    PASSTHROUGH_SERVO_STATES.Ready :                    // Keep track    
                                                        IF jogInPB THEN
															passthroughSetpoint := 2.0 + HMIData.passthroughOffset;
															capturePassthroughPos := passthroughPosition;
															state := PASSTHROUGH_SERVO_STATES.MovePassthroughIn;
														ELSIF jogOutPB THEN
															passthroughSetpoint := 8.0 + HMIData.passthroughOffset;
															capturePassthroughPos := passthroughPosition;
															state := PASSTHROUGH_SERVO_STATES.MovePassthroughOut;
														ELSIF jogInONS.OSF OR jogOutONS.OSF THEN
															Globals.passthroughChangedFromJog := TRUE;
															pressureBarEndStopMotor.Stop();
														END_IF
														
                                                        IF _movePassthrough THEN
															passthroughTravel := ABS(passthroughPosition - (passthroughSetpoint + HMIData.passthroughOffset));
                                                            IF mustMovePassthroughOut THEN
                                                                state := PASSTHROUGH_SERVO_STATES.MovePassthroughOut;
                                                                ELSE state := PASSTHROUGH_SERVO_STATES.MovePassthroughIn;
                                                            END_IF
                                                        END_IF
                                                        IF _homeEndStop THEN
                                                            state := PASSTHROUGH_SERVO_STATES.StartHoming;
                                                        END_IF
    
    PASSTHROUGH_SERVO_STATES.Fault :   					pressureBarEndStopMotor.Stop();        
END_CASE

METHOD MovePassthrough
VAR_INPUT
    PassthroughSetting : REAL;
END_VAR
passthroughSetpoint := PassthroughSetting;
mustMovePassthroughOut := (passthroughSetpoint > passthroughPosition);
_movePassthrough := TRUE;
END_METHOD

PROPERTY Ready : BOOL
GET
Ready := _ready;
END_GET
SET
_ready := Ready;
END_SET
END_PROPERTY

PROPERTY Mode : DEVICE_MODES
GET
Mode := _mode;
END_GET
SET
_mode := Mode;
END_SET
END_PROPERTY

METHOD AckRequest
VAR_INPUT
END_VAR
_ackRequest := TRUE;
END_METHOD

METHOD HomeEndStop
VAR_INPUT
END_VAR
_homeEndStop := TRUE;
END_METHOD

END_FUNCTION_BLOCK

// FBs/Cylinders/FB_CylinderFaults
FUNCTION_BLOCK FB_CylinderFaults
VAR_INPUT
	enable : BOOL;
	extendCommand : BOOL;
	extendedInput : BOOL;
	retractCommand : BOOL;
	retractedInput : BOOL;
	faultTime : TIME := T#2500ms;
END_VAR
VAR_OUTPUT
	failToExtend : BOOL;
	failToRetract : BOOL;
END_VAR
VAR
	extendFaultTimer : Standard.TON;
	retractFaultTimer : Standard.TON;
END_VAR
VAR_IN_OUT
END_VAR

extendFaultTimer(PT := faultTime, Q => failToExtend);
retractFaultTimer(PT := faultTime, Q => failToRetract);
IF enable THEN
	IF extendCommand THEN
		retractFaultTimer.IN := FALSE;
		extendFaultTimer.IN := NOT extendedInput;
	ELSIF retractCommand THEN
		extendFaultTimer.IN := FALSE;
		retractFaultTimer.IN := NOT retractedInput;
	ELSE
		retractFaultTimer.IN := FALSE;
		extendFaultTimer.IN := FALSE;
	END_IF
ELSE
	retractFaultTimer.IN := FALSE;
	extendFaultTimer.IN := FALSE;
END_IF

END_FUNCTION_BLOCK

// FBs/FB_HMILight
FUNCTION_BLOCK FB_HMILight
VAR_INPUT
END_VAR
VAR_OUTPUT
	lightOutput : BOOL;
END_VAR
VAR
	_turnOn : BOOL;
	_blinkFast : BOOL;
	_blinkSlow : BOOL;
	blinker : OSCAT_BASIC.PWM_DC := (F := 1, DC := 0.5);
	slowBlinkSec : REAL := 1;
	fastBlinkSec : REAL := 0.5;
END_VAR

IF _blinkFast THEN
	blinker.F := fastBlinkSec;
ELSIF _blinkSlow THEN 
	blinker.F := slowBlinkSec;
END_IF
	
blinker(F:= , DC:= , Q=> );

lightOutput := _turnOn OR (blinker.Q AND (_blinkFast OR _blinkSlow));

METHOD BlinkSlow
VAR_INPUT
END_VAR
_blinkFast := FALSE;
_blinkSlow := TRUE;
_turnOn := FALSE;
END_METHOD

METHOD BlinkFast
VAR_INPUT
END_VAR
_blinkFast := TRUE;
_blinkSlow := FALSE;
_turnOn := FALSE;
END_METHOD

METHOD TurnOff
VAR_INPUT
END_VAR
_blinkFast := FALSE;
_blinkSlow := FALSE;
_turnOn := FALSE;
END_METHOD

METHOD TurnOn
VAR_INPUT
END_VAR
_blinkFast := FALSE;
_blinkSlow := FALSE;
_turnOn := TRUE;
END_METHOD

END_FUNCTION_BLOCK

// FBs/Components/FillerFB
FUNCTION_BLOCK FillerFB EXTENDS BaseComponentFB IMPLEMENTS IComponentStatus
VAR_INPUT
	fillerTrigger : BOOL;
	activateFiller : BOOL;
	fillerOK : BOOL;
	dropTime : REAL;
END_VAR
VAR_OUTPUT
	state : FILLER_STATES;
	fillerModeActive : BOOL;
	waitingForFiller : BOOL;
	cycleBagRequest : BOOL;
	cycleBaggerToActivateFiller : Warning;
	notReady : FB_Fault(name := 'Not Ready');
END_VAR
VAR
	_baggerCycleInitiated : BOOL;
    _baggerCycledAndReady : BOOL;
	fillerRequestedCycle : BOOL;
	fillerTrigONS : FB_ONS;
	dropTimer : Standard.TON;
END_VAR
	
VAR_IN_OUT
END_VAR

//    Function Block: FillerFB
//    Description: Filler state machine
//    Created by: Ben Hess
//    Created Date: October 16th, 2019
SUPER^();
dropTimer(PT := TO_TIME(dropTime * 1000));
IF resetONS.Q OR HMIData.faultActive OR NOT enable OR NOT activateFiller THEN
	state := FILLER_STATES.Idle;
	fillerRequestedCycle := FALSE;
	cycleBaggerToActivateFiller.active := FALSE;
	waitingForFiller := FALSE;
	cycleBagRequest := FALSE;
	_baggerCycledAndReady := FALSE;
	_baggerCycleInitiated := FALSE;
	dropTimer.IN := FALSE;
END_IF

IF NOT fillerOK AND enable AND activateFiller THEN
	notReady.Trigger();
END_IF

fillerTrigONS(CLK := fillerTrigger);
IF fillerTrigONS.OSR THEN
	fillerRequestedCycle := TRUE;
END_IF

CASE state OF
	FILLER_STATES.Idle :							IF (activateFiller AND enable) AND NOT HMIData.faultActive THEN
														state := FILLER_STATES.CycleBaggerToActiveFiller;
													END_IF
	
	FILLER_STATES.CycleBaggerToActiveFiller :		// Operator must cycle a bag out first to guarentee bag open and ready for filler
													cycleBaggerToActivateFiller.active := TRUE;
													
													IF _baggerCycledAndReady THEN
														cycleBaggerToActivateFiller.active := FALSE;
														_baggerCycledAndReady := FALSE;
														fillerRequestedCycle := FALSE;
														state := FILLER_STATES.WaitingForFiller;
													END_IF
	
	FILLER_STATES.WaitingForFiller :				// Waiting for filler trigger to initiate cycle
													waitingForFiller := TRUE;
													IF fillerRequestedCycle THEN
														waitingForFiller := FALSE;	
														//IF NOT HMIData.baggerInhibited.active THEN
															fillerRequestedCycle := FALSE;
															state := FILLER_STATES.Dropping;	
														//END_IF
													END_IF
													
	FILLER_STATES.Dropping :						// Filler is dropping product
													dropTimer.IN := TRUE;
													IF dropTimer.Q THEN
														IF NOT HMIData.baggerInhibited.active THEN
															dropTimer.IN := FALSE;
															cycleBagRequest := TRUE;
															state := FILLER_STATES.BaggerCycling;	
														END_IF
													END_IF
	
	FILLER_STATES.BaggerCycling :					// Wait for bag to open 
													IF _baggerCycleInitiated THEN
														_baggerCycleInitiated := FALSE;
														cycleBagRequest := FALSE;
													END_IF
													
													IF _baggerCycledAndReady THEN
														_baggerCycledAndReady := FALSE;
														state := FILLER_STATES.WaitingForFiller;
													END_IF
	
	FILLER_STATES.Fault :
	
END_CASE

METHOD BaggerCycledAndReady : BOOL
VAR_INPUT
END_VAR
_baggerCycledAndReady := TRUE;
END_METHOD

PROPERTY Ready : BOOL
SET
_ready := Ready;
END_SET
GET
Ready := _ready;
END_GET
END_PROPERTY

METHOD BaggerCycleInitiated : BOOL
VAR_INPUT
END_VAR
_baggerCycleInitiated := TRUE;
END_METHOD

PROPERTY Mode : DEVICE_MODES
SET
_mode := Mode;
END_SET
GET
Mode := _mode;
END_GET
END_PROPERTY

METHOD Reset : BOOL
VAR_INPUT
END_VAR
SUPER^.Reset();
END_METHOD

END_FUNCTION_BLOCK

// FBs/Components/MurrIOFB
FUNCTION_BLOCK MurrIOFB EXTENDS BaseComponentFB IMPLEMENTS IComponentStatus
VAR_INPUT
	headNodeEnabled : BOOL;
	guardNodeEnabled : BOOL;
	printerNodeEnabled : BOOL;
	dischargeNodeEnabled : BOOL;
	auxIONodeEnabled : BOOL;
	configVersion : CONFIG_VERSIONS;
	ptrMachineOptionsManagementOutputs : POINTER TO BYTE;
	ptrSystemStatusInputs : POINTER TO BYTE;
END_VAR
VAR_OUTPUT
	commFailController : FB_Fault(name := 'Communication Fail - Bus Master to Controller');
	commFailNode : FB_Fault(name := 'Communication Fail - Bus Master to I/O Node');
	configActive : Warning;	// I/O Configuration Active, please wait
	ok : BOOL; 		// I/O Configuration and Communication good
END_VAR
VAR
	systemStatusINT : INT;
	systemStatusState : MURR_SYSTEM_STATES;
	MOMConfigLast : BYTE;
	restartBusnodePulse : MonostableMultivibratorFB;
END_VAR
	
VAR_IN_OUT

END_VAR

//    Function Block: MurrIOFB
//    Description: Alarms, faults, configuration of the Murr Cube67+ Bus Node
//    Created by: Ben Hess
//    Created Date: October 16th, 2019
SUPER^();

// Set bit 33 to true for 1 second to reset nodes
restartBusnodePulse.DwellSetting := 1000;
restartBusnodePulse(Q => ptrMachineOptionsManagementOutputs[4].1);

// Exit this FB if invaild pointers set
IF ptrMachineOptionsManagementOutputs = 0 OR ptrSystemStatusInputs = 0 THEN
	RETURN;
END_IF

// MOM config - MOM bits are counted from Slot 001 to 4xx and are counted based on the "Maximium" configuration hard coded in the bus master
// Here we can select which verison of code we have in order to utilize MOM correctly if we add additional modules in the future.
CASE configVersion OF
	CONFIG_VERSIONS.V_1_1 :		//
									ptrMachineOptionsManagementOutputs[0].0 := NOT headNodeEnabled;
									ptrMachineOptionsManagementOutputs[0].1 := NOT guardNodeEnabled;
									ptrMachineOptionsManagementOutputs[0].2 := NOT dischargeNodeEnabled;
									ptrMachineOptionsManagementOutputs[0].3 := NOT printerNodeEnabled;
									ptrMachineOptionsManagementOutputs[0].4 := FALSE;
									
								

	CONFIG_VERSIONS.V_1_2, CONFIG_VERSIONS.V_1_3,CONFIG_VERSIONS.V_1_4 : 		// Added aux IO to 1.2 and BCV trigger to 1.3
									ptrMachineOptionsManagementOutputs[0].0 := NOT headNodeEnabled;
									ptrMachineOptionsManagementOutputs[0].1 := NOT guardNodeEnabled;
									ptrMachineOptionsManagementOutputs[0].2 := NOT auxIONodeEnabled;
									ptrMachineOptionsManagementOutputs[0].3 := NOT dischargeNodeEnabled;
									ptrMachineOptionsManagementOutputs[0].4 := NOT printerNodeEnabled;
END_CASE


// Run config if IO bus node is waiting on config
systemStatusINT := ptrSystemStatusInputs^;
systemStatusState := systemStatusINT;

// Prevent a IO node reset on boot for no reason
IF Globals.firstScan THEN
	MOMConfigLast := ptrMachineOptionsManagementOutputs[0];
END_IF

// Trigger fault for node not present, or node seen where one shouldn't be 
IF systemStatusState = MURR_SYSTEM_STATES.No_Comm_To_Configured_Node THEN
	commFailNode.Trigger();
END_IF

// A 0 at system state indicates comm fail to controller
IF systemStatusState = 0 THEN
	commFailController.Trigger();
END_IF

// Alert user to MOM config active
IF systemStatusState = MURR_SYSTEM_STATES.Waiting_For_MOM OR
	systemStatusState = MURR_SYSTEM_STATES.Configuring_MOM OR
	systemStatusState = MURR_SYSTEM_STATES.Internal_Comm_Disabled
THEN
	configActive.active := TRUE;
ELSE
	configActive.active := FALSE;
END_IF

// I/O Block is OK only in this state, otherwise we can't trust any I/O coming back
ok := (systemStatusState = MURR_SYSTEM_STATES.Internal_Comm_OK);

CASE systemStatusState OF

	
	MURR_SYSTEM_STATES.Waiting_For_MOM: 			// Bit 32 is Configure MOM bit
													ptrMachineOptionsManagementOutputs[4].0 := TRUE;
													ptrMachineOptionsManagementOutputs[4].1 := FALSE;
													
	
	MURR_SYSTEM_STATES.Configuring_MOM : 			//
													ptrMachineOptionsManagementOutputs[4].0 := FALSE;
													
											

														
											
ELSE
													ptrMachineOptionsManagementOutputs[4].0 := FALSE;
													//IF config changes here, send it down after restarting
													IF ptrMachineOptionsManagementOutputs[0] <> MOMConfigLast THEN
														restartBusnodePulse.Trigger();
														MOMConfigLast := ptrMachineOptionsManagementOutputs[0];
													END_IF
END_CASE

PROPERTY Mode : DEVICE_MODES
GET
Mode := _mode;
END_GET
SET
_mode := Mode;
END_SET
END_PROPERTY

PROPERTY Ready : BOOL
GET
Ready := _ready;
END_GET
SET
_ready := Ready;
END_SET
END_PROPERTY

END_FUNCTION_BLOCK

// FBs/Components/FunnelFB
FUNCTION_BLOCK FunnelFB EXTENDS BaseComponentFB
VAR_INPUT
	sensorsInstalled : BOOL;							// Are open/closed sensors installed?
	openSensor : BOOL;									// Open sensor input
	closedSensor : BOOL;								// Closed sensor input
END_VAR	
VAR_OUTPUT
	opened : BOOL;										// Funnel Opened status
	closed : BOOL;										// Funnel Closed status
	closeOutput : BOOL;									// Map to physical close output
	openOutput : BOOL;									// Map to physical open output
	failToOpen : FB_Fault(name := 'Failed to Open');	// Failed to Open fault
	failToClose : FB_Fault(name := 'Failed to Close');	// Failed to Close fault
END_VAR
VAR
	_delayTimeInMS : UINT; 								// Delay before open in mS
	_closeReq : BOOL;									// Close reqested from CloseNow()
	_openReq : BOOL;									// Open requested from OpenNow()
	openDelayTimer : Standard.TON;						// Open delay timer
	openingTimer : Standard.TON;						// Opening timer
	closingTimer : Standard.TON;						// Closing timer
	faultTimer : FB_CylinderFaults;						// Fault timer for open/close faults
END_VAR

//    Function Block: FunnelFB
//    Description: Funnel
//    Created by: Ben Hess
//    Created Date: November 18th, 2019

IF _reset THEN
	_openReq := FALSE;
	_closeReq := FALSE;
	openingTimer.IN := FALSE;
	closingTimer.IN := FALSE;
	openDelayTimer.IN := FALSE;
END_IF

// Setup timers
openDelayTimer();
openingTimer();
closingTimer();

// Use opening/closing timers for debounce if sensors enabled
// or for actual opening/closing time after command to move if disabled
IF sensorsInstalled THEN
	openingTimer.IN := openSensor;
	closingTimer.IN := closedSensor;
ELSE
	openingTimer.IN := openOutput;
	closingTimer.IN := closeOutput;
END_IF

// Set open/closed status of funnel
opened := openingTimer.Q;
closed := closingTimer.Q;


// Set physical outputs depending on command
IF enable THEN
	IF _closeReq THEN
		closeOutput := TRUE;
		openOutput := FALSE;
		_closeReq := FALSE;
	ELSIF _openReq THEN
		openDelayTimer.IN := TRUE;
		closeOutput := FALSE;
		openOutput := openDelayTimer.Q;
		_openReq := FALSE;
	END_IF
ELSE
	// Turn everything off if disabled
	closeOutput := FALSE;
	openOutput := FALSE;
	_openReq := FALSE;
	_closeReq := FALSE;
	openingTimer.IN := FALSE;
	closingTimer.IN := FALSE;
	openDelayTimer.IN := FALSE;
END_IF

// Fault timer for failed to reach open/closed sensors
faultTimer(
	enable:= THIS^.enable AND sensorsInstalled, 
	extendCommand:= closeOutput, 
	extendedInput:= closedSensor, 
	retractCommand:= openOutput, 
	retractedInput:= openSensor, 
	faultTime:= T#1S, 
	failToExtend=> failToClose.faultTrigger, 
	failToRetract=> failToOpen.faultTrigger);
	
SUPER^();

PROPERTY DelaySetting : REAL
GET
DelaySetting := TO_REAL(openDelayTimer.PT ) / 1000;
END_GET
SET
openDelayTimer.PT := TO_TIME(DelaySetting * 1000);
END_SET
END_PROPERTY

METHOD CloseNow : BOOL
VAR_INPUT
END_VAR
_closeReq := TRUE;
END_METHOD

PROPERTY OpeningTime : REAL
SET
openingTimer.PT := TO_TIME(OpeningTime * 1000);
END_SET
GET
OpeningTime := TO_REAL(openingTimer.PT) / 1000;
END_GET
END_PROPERTY

METHOD OpenNow : BOOL
VAR_INPUT
END_VAR
_openReq := TRUE;
END_METHOD

PROPERTY ClosingTime : REAL
GET
ClosingTime := TO_REAL(closingTimer.PT) / 1000;
END_GET
SET
closingTimer.PT := TO_TIME(ClosingTime * 1000);
END_SET
END_PROPERTY

END_FUNCTION_BLOCK

// FBs/Components/BarcodeReaderFB
FUNCTION_BLOCK BarcodeReaderFB EXTENDS BaseComponentFB
VAR_INPUT
	feedSpeed : REAL;
	positionOffset : REAL;
	distanceToScan : REAL;
	readGoodInput : BOOL;
	badReadFaultCountSetting : UDINT;
END_VAR	
VAR_OUTPUT
	triggerScannerOutput : BOOL;
	xBusy : BOOL;
	xDone : BOOL;
	currentGoodReadCount : UDINT;
	currentBadReadCount : UDINT;
	barcodeFault : BOOL;
END_VAR
VAR
	_goodRead : BOOL;
	_badread : BOOL;
	_trigger : BOOL;
	state : BCR_STATES;
	waitForReadTimer : Standard.TON;
	positionOffsetDelay : Standard.TON;
END_VAR
VAR CONSTANT
	MILLISECONDS_IN_SECOND : INT := 1000;
END_VAR

//    Function Block: BarcodeReaderFB
//    Description: Trigger the barcode verifier and receive a "Barcode OK" signal, or nothing which indicates no read.
//    Created by: Ben Hess
//    Created Date: January 29th, 2020

// Setup timers for reading offset and scanning distance
IF positionOffset > 0 THEN
	positionOffsetDelay(PT := TO_TIME(MILLISECONDS_IN_SECOND / (feedSpeed / positionOffset)) + T#120ms);
ELSE
	positionOffsetDelay(PT := T#0S);
END_IF

IF distanceToScan > 0 THEN
	waitForReadTimer(PT := TO_TIME(MILLISECONDS_IN_SECOND / (feedSpeed / distanceToScan)));
ELSE
	waitForReadTimer(PT := T#0S);
END_IF

IF _reset OR NOT enable THEN
	//
	state := BCR_STATES.Idle;
	barcodeFault := FALSE;
END_IF

CASE state OF
	
	BCR_STATES.Idle:				// Wait for trigger
									triggerScannerOutput := FALSE;
									waitForReadTimer.IN := FALSE;
									positionOffsetDelay.IN := FALSE;
									
									xBusy := FALSE;
									IF _trigger THEN
										state := BCR_STATES.WaitForOffset;
										positionOffsetDelay.IN := TRUE;
										xBusy := TRUE;
										xDone := FALSE;
									END_IF
									
									_trigger := FALSE;
									
	BCR_STATES.WaitForOffset: 		// Wait for offset to trigger read
									IF positionOffsetDelay.Q THEN
										state := BCR_STATES.TriggerReader;
										positionOffsetDelay.IN := FALSE;
									END_IF
									
	BCR_STATES.TriggerReader:		// Trigger the reader and then move to waiting state for result
									triggerScannerOutput := TRUE;
									waitForReadTimer.IN := TRUE;
									state := BCR_STATES.WaitingForResult;
									
	
	BCR_STATES.WaitingForResult:	// Wait for delayToCheckReadStatus timer.  If it times out we did not get a good read
									IF readGoodInput THEN
										_goodRead := TRUE;
										_badread := FALSE;
										currentGoodReadCount := currentGoodReadCount + 1;
										currentBadReadCount := 0;
										xDone := TRUE;
										state := BCR_STATES.Idle;
									ELSIF waitForReadTimer.Q THEN
										_goodRead := FALSE;
										_badread := TRUE;
										currentGoodReadCount := 0;
										currentBadReadCount := currentBadReadCount + 1;
										IF badReadFaultCountSetting > 0 THEN
											IF currentBadReadCount >= badReadFaultCountSetting THEN
												barcodeFault := TRUE;
											END_IF
										END_IF
										xDone := TRUE;
										state := BCR_STATES.Idle;
									END_IF
	
	BCR_STATES.Resetting:
	
END_CASE

SUPER^();

METHOD Trigger : BOOL
VAR_INPUT
END_VAR
_trigger := TRUE;
END_METHOD

PROPERTY BadRead : BOOL
SET
END_SET
GET
END_GET
END_PROPERTY

PROPERTY GoodRead : BOOL
GET
END_GET
SET
END_SET
END_PROPERTY

END_FUNCTION_BLOCK

// FBs/Components/KeyenceL20FB/KeyenceNL20FB
FUNCTION_BLOCK KeyenceNL20FB EXTENDS BaseComponentFB IMPLEMENTS IComponentStatus
VAR_INPUT
	ptrEIPInputs : POINTER TO WORD;
	ptrEIPOutputs : POINTER TO WORD;
	triggerInput : BOOL;
END_VAR
VAR_OUTPUT
	lastReadData : STRING[100];
	xBusy : BOOL;
	xDone : BOOL;
	goodRead : BOOL;
	badRead : BOOL;
END_VAR
VAR
	error : BOOL;
	readDataUpdateAvailable : BOOL;
	readDataUpdateComplete : BOOL;
	bufferOverflowError : BOOL;
	generalError : BOOL;
	bcvBusy : BOOL;
	readingComplete : BOOL;
	in1Status : BOOL;
	in2Status : BOOL;
	out1Status : BOOL;
	out2Status : BOOL;
	out3Status : BOOL;
	out4Status : BOOL;
	errorCode : UINT;
	readDataReadyCount : UINT;
	readDataUpdateCount : UINT;
	readDataLength : UINT;
	readData : POINTER TO STRING[100];
	
	readDataUpdatePermitted : BOOL;
	errorAndBufferClear : BOOL;
	readingStartRequest : BOOL;
	readingCompleteAck : BOOL;
	bankNumber : UINT;
	
	state : eKeyenceLN20FB_States;
	triggerONS : FB_ONS;
	readingCompleteTrigger : MonostableMultivibratorFB();
END_VAR
	
VAR_IN_OUT

END_VAR

//    Function Block: KeyenceL20FB
//    Description: Alarms, faults, configuration of the Keyence L-N20 barcode scanner base
//    Created by: Ben Hess
//    Created Date: Feb 28th, 2020


// Exit FB if pointers are invalid
IF ptrEIPInputs = 0 OR ptrEIPOutputs = 0 THEN
	RETURN;
END_IF
triggerONS(CLK := triggerInput);

readingCompleteTrigger.DwellSetting := 500;
readingCompleteTrigger(Q => readingCompleteAck);
// Map statuses to friendly variables
error := ptrEIPInputs[0].0;
readDataUpdateAvailable := ptrEIPInputs[0].1;
readDataUpdateComplete := ptrEIPInputs[0].2;
bufferOverflowError := ptrEIPInputs[0].6;
generalError := ptrEIPInputs[0].7;
bcvBusy := ptrEIPInputs[0].8;

readingComplete := ptrEIPInputs[1].0;

in1Status := ptrEIPInputs[2].0;
in2Status := ptrEIPInputs[2].1;
out1Status := ptrEIPInputs[2].4;
out2Status := ptrEIPInputs[2].5;
out3Status := ptrEIPInputs[2].6;
out4Status := ptrEIPInputs[2].7;

errorCode := ptrEIPInputs[16];

readDataReadyCount := ptrEIPInputs[18];
readDataUpdateCount := ptrEIPInputs[19];

readDataLength := ptrEIPInputs[21];
readData := ADR(ptrEIPInputs[22]);


IF resetONS.Q THEN
	state := eKeyenceLN20FB_States.Reset;
END_IF



CASE state OF
	eKeyenceLN20FB_States.Idle: 			//
											IF readingComplete THEN
													readingCompleteTrigger.Trigger();
												END_IF
											IF triggerONS.OSR THEN
												readingStartRequest := TRUE;
												xBusy := TRUE;
												xDone := FALSE;
												badRead := FALSE;
												goodRead := FALSE;
												lastReadData := '---Read in Progress---';
												state := eKeyenceLN20FB_States.WaitForStatus;
											END_IF

	eKeyenceLN20FB_States.WaitForStatus:	//
											IF readingComplete OR NOT triggerInput THEN
												state := eKeyenceLN20FB_States.SetStatus;
												readingStartRequest := FALSE;
												IF readingComplete THEN
													readingCompleteTrigger.Trigger();
												END_IF
												
											END_IF
	
	eKeyenceLN20FB_States.SetStatus:		// Set the current read status and string
											// If trigger input goes away or barcode error seen set bad read
											IF NOT triggerInput OR out2Status THEN
												badRead := TRUE;
												goodRead := FALSE;
												state := eKeyenceLN20FB_States.WaitForReadClear;
												IF out2Status THEN
													lastReadData := '---BAD READ---';
												ELSE
													lastReadData := '---NO READ---';
												END_IF
											ELSIF out1Status THEN
												goodRead := TRUE;
												badRead := FALSE;
												// Strip terminating char (0x0D) from string to get clean read barcode
												lastReadData := LEFT(readData^, readDataLength - 1);
												state := eKeyenceLN20FB_States.WaitForReadClear;
											END_IF
											
	eKeyenceLN20FB_States.WaitForReadClear:	//
											IF readingComplete THEN
												readingCompleteTrigger.Trigger();
											END_IF
											IF NOT readingComplete THEN
												xBusy := FALSE;
												xDone := TRUE;
												state := eKeyenceLN20FB_States.Idle;
											END_IF 									

	eKeyenceLN20FB_States.Reset: 			//
											IF readingComplete THEN
												readingCompleteTrigger.Trigger();
											END_IF
											
												readingStartRequest := FALSE;
												xBusy := FALSE;
												xDone := FALSE;
												badRead := FALSE;
												goodRead := FALSE;
												state := eKeyenceLN20FB_States.Idle;
											
END_CASE	

// Outputs to barcode verifier
ptrEIPOutputs[0].1 :=  readDataUpdatePermitted;
ptrEIPOutputs[0].7 :=  errorAndBufferClear;
ptrEIPOutputs[0].8 := readingStartRequest;
ptrEIPOutputs[1].0 := readingCompleteAck;
ptrEIPOutputs[2] := bankNumber;

// Call to super FB.
SUPER^();

PROPERTY Ready : BOOL
SET
_ready := Ready;
END_SET
GET
Ready := _ready;
END_GET
END_PROPERTY

PROPERTY Mode : DEVICE_MODES
SET
_mode := Mode;
END_SET
GET
Mode := _mode;
END_GET
END_PROPERTY

END_FUNCTION_BLOCK

// FBs/Components/EZFeedFB/EZFeedFB
FUNCTION_BLOCK EZFeedFB EXTENDS BaseComponentFB IMPLEMENTS IComponentStatus
VAR_INPUT
	baggerFaulted : BOOL;
	enableEZFeed : BOOL;					// Enable EZFeed conveyor (In Use)
	continuousModeEnable : BOOL; 			// 0 = indexing mode, 1 = continuous mode
	partsCountingModeEnable : BOOL;			// 0 = Flight counting only, 1 = Parts counting (requires sensor or light curtains)
	flightPresentSensor : BOOL;				// Flight present 
	partPresentSensor : BOOL;				// Part present/dropping (photoeye, light curtain, etc)
	waitingForFiller : BOOL;				// Waiting for Filler signal from bagger
	indexDwellSetting : REAL;				// Indexing dwell setting
	flightTarget : DINT;					// For Flight counting mode, target flights before starting cycle
	partsTarget : DINT;						// For Parts counting mode, target parts before starting cycle
	emptyPartsWarningSetting : DINT;		// For Parts counting mode, setting of empty flights counted before warning issued
	restartFromEmptyParts : BOOL;			// Restart EZFeed after starvation/empty parts. Usually cycle start button
END_VAR
VAR_OUTPUT
	state : EZFEED_STATES;					// State machine
	runVFD : BOOL;							// Run VFD output
	flightCount : DINT;						// Actual flight count
	partsCount : DINT;						// Actual parts count
	emptyPartsWarningCount : DINT;			// Actual empty flights count
	EZFeedDone : BOOL;						// EZFeed done - cycle bagger
	emptyPartsWarning : BOOL;				// Parts starved
END_VAR
VAR
	indexDwellTimer : TON;
	flightPresentONS : FB_ONS;
	partPresentONS : FB_ONS;
END_VAR
	
VAR_IN_OUT
END_VAR

//    Function Block: EZFeedFB
//    Description: EZFeed state machine
//    Created by: Ben Hess
//    Created Date: December 3rd, 2020


// Run parent FB
SUPER^();

// Resetting 
IF resetONS.Q OR baggerFaulted OR NOT enable OR NOT enableEZFeed THEN
	state := EZFEED_STATES.Idle;
	runVFD := FALSE;
	EZFeedDone := FALSE;
	flightCount := 0;
	partsCount := 0;
	emptyPartsWarningCount := 0;
END_IF

// Timer for indexing dwell
indexDwellTimer(PT := TO_TIME(indexDwellSetting * 1000), IN := state = EZFEED_STATES.IndexDwell);

flightPresentONS(CLK := flightPresentSensor);
partPresentONS(CLK := partPresentSensor);

// Parts Counting logic
IF partsCountingModeEnable AND (state = EZFEED_STATES.IndexingFlightMode OR state = EZFEED_STATES.IndexDwell) THEN
	// Count flights for empty parts watchdog timer
	IF flightPresentONS.OSR THEN
		emptyPartsWarningCount := emptyPartsWarningCount + 1;
	END_IF
	
	IF partPresentONS.OSF THEN
		emptyPartsWarningCount := 0;
		partsCount := partsCount + 1;
	END_IF
	
END_IF

CASE state OF
	
	EZFEED_STATES.Idle :						// When filler reports as waiting for filler, start indexing the EZFeed
												IF enableEZFeed AND waitingForFiller THEN
													IF partsCountingModeEnable THEN
														state := EZFEED_STATES.IndexingPartsMode;
													ELSE
														state := EZFEED_STATES.IndexingFlightMode;
													END_IF
													
												END_IF
	
	EZFEED_STATES.IndexingPartsMode :			// Check parts count and start bagger if count reached
												IF partsCount >= partsTarget THEN
													partsCount := 0;
													runVFD := FALSE;
													EZFeedDone := TRUE;
													state := EZFEED_STATES.WaitForBaggerCycleComplete;
												ELSE
													// Dwell at each flight for indexing mode
													IF NOT continuousModeEnable THEN
														runVFD := FALSE;
														state := EZFEED_STATES.IndexDwell;
													END_IF
												END_IF

												
		
	EZFEED_STATES.IndexingFlightMode :			// Run the VFD until flight seen. Keep going until target reached in Continuous mode or stop for dwell time in indexing mode
												runVFD := TRUE;
												IF flightPresentONS.OSR THEN
													flightCount := flightCount + 1;
													// Check flight count and start bagger if count reached
													IF flightCount >= flightTarget THEN
														runVFD := FALSE;
														EZFeedDone := TRUE;
														flightCount := 0;
														state := EZFEED_STATES.WaitForBaggerCycleComplete;
													ELSE
														// Dwell at each flight for indexing mode
														IF NOT continuousModeEnable THEN
															runVFD := FALSE;
															state := EZFEED_STATES.IndexDwell;
														END_IF
													END_IF
												END_IF
												
	EZFEED_STATES.IndexDwell :					// Dwell at each flight for indexing mode
												IF indexDwellTimer.Q THEN
													IF partsCountingModeEnable THEN
														IF partsCount >= partsTarget THEN
															partsCount := 0;
															EZFeedDone := TRUE;
															state := EZFEED_STATES.WaitForBaggerCycleComplete;
														ELSE
															state := EZFEED_STATES.IndexingPartsMode;
														END_IF
													ELSE
														state := EZFEED_STATES.IndexingFlightMode;
													END_IF
												END_IF
												
	EZFEED_STATES.WaitForBaggerCycleComplete :	// Once bagger cycle is complete then resume indexing
												IF waitingForFiller THEN
													IF partsCountingModeEnable THEN
														state := EZFEED_STATES.IndexingPartsMode;
													ELSE
														state := EZFEED_STATES.IndexingFlightMode;
													END_IF
												END_IF
								
	EZFEED_STATES.PartsStarved:					//
												
									
	EZFEED_STATES.Fault :						//
												

END_CASE

PROPERTY Mode : DEVICE_MODES
SET
_mode := Mode;
END_SET
GET
Mode := _mode;
END_GET
END_PROPERTY

PROPERTY Ready : BOOL
GET
Ready := _ready;
END_GET
SET
_ready := Ready;
END_SET
END_PROPERTY

METHOD Reset : BOOL
VAR_INPUT
END_VAR
SUPER^.Reset();
END_METHOD

END_FUNCTION_BLOCK

// FBs/GetTime
FUNCTION_BLOCK GetTime
VAR_INPUT
END_VAR
VAR_OUTPUT
    currentDateAndTime : DATE_AND_TIME;
    
END_VAR
VAR
    iState                    : INT;
    udiUtcTime             : UDINT;
    udiUtcTimeLocal     : UDINT;
    strTimeDate         : SYSTIMEDATE;
    strTimeDateLocal     : SYSTIMEDATE;
    dtDateTimeUTC        : DATE_AND_TIME;
    timeLeftTime        : TIME;
    timeLeftDWORD        : DWORD;
    dDateUTC            : DATE;
    todTimeOfDayUTC        : TOD;
    
    tSysStartTime        : TIME;
    systimeStartNano    : SYSTIME;
    udiStartTimeResult    : UDINT;
    
    udiResult             : UDINT;
    
    
    GetDateAndTime            : DTU.GetDateAndTime;
    SetTimeZoneInformation    : DTU.SetTimeZoneInformation;
    
    dtCurrent                : DATE_AND_TIME;
    dtConcated                : DATE_AND_TIME;
    eWeekday                 : RTCLK.WEEKDAY;
    uiYear                     : UINT;
    uiMonth                     : UINT;
    uiDay                     : UINT;
    uiHour                     : UINT;
    uiMinute                 : UINT;
    uiSecond                 : UINT;
        
    dtuError                : DTU.ERROR;
END_VAR

CASE iState OF

    0:    
        iState:= 1;
        
    1:  // retrieves the target date and time, including the timezone information which was set before
        GetDateAndTime( xExecute:= TRUE);
        IF GetDateAndTime.xDone THEN
            dtCurrent:= GetDateAndTime.dtDateAndTime;
            GetDateAndTime(xExecute:= FALSE);
			currentDateAndTime := dtCurrent;
            //timeLeft := TIME_TO_DT(DT_TO_TIME(targetDate) - DT_TO_TIME(dttarget));
            iState:= 2;
        END_IF
        IF GetDateAndTime.xError THEN
            GetDateAndTime(xExecute:= FALSE);
            iState:= 32767;
        END_IF
    
    2: (*set a spedific date and time --> returns a variable of type DATE_AND_TIME 
         DateConcat --> set only date information --> returns a variable of type DATE
         TODConcat  --> set only the time information  --> returns a variable of TOD (Time of day) *)
        IF dtuError = 0 THEN
            iState := 3;
        ELSE
            iState := 32767;
        END_IF
        
    3:  (*a DATE_AND_TIME variable is splitted in its parts, like year, month, day etc.
            DateSplit --> the same function for a DATE variable
            TODSplit  --> the same function for a TOD variable *)

            
        IF dtuError = 0 THEN
            iState:= 1;
        ELSE
            iState:= 32767;
        END_IF
        
    32767: ; //error

END_CASE

END_FUNCTION_BLOCK

// FBs/FunctionalAreas/FB_MOABHead_Electric
FUNCTION_BLOCK FB_MOABHead_Electric EXTENDS BaseComponentFB
VAR_INPUT
    motorizedSealFlattenersMode : DEVICE_MODES := DEVICE_MODES.Auto;
    electricPressureBarMode : DEVICE_MODES := DEVICE_MODES.Auto;
	vacuumPickerMode : DEVICE_MODES;
    startCycle : BOOL;
    bagDeliveryMode : DEVICE_MODES;        // Mode of bag delivery system
    printerMode : DEVICE_MODES;        // Mode of printer
	passthroughMode : DEVICE_MODES;
    batchSetting : DINT;            // Batch setpoint
    batchCount : DINT;                // Actual batch cycles
    enableBatch : BOOL;                // Enable Batch Mode
    enableBatchONS : F_TRIG;
	passthroughSetting : REAL;
    passthroughSettingLast : REAL;
	bagDropDelay : UINT := 1000;
END_VAR
VAR_OUTPUT
    readyToRun : BOOL;
    state : HEAD_STATES;
    sealAndSeparateSubState : SEAL_SEPARATE_STATES;
    releaseAndFeedSubState : RELEASE_FEED_STATES;
    openBagSubState : BAG_OPEN_ASSIST_STATES;
	finishCycleSubState : FINISH_CYCLE_STATES;
END_VAR
VAR
    motorizedSealFlatteners : MotorizedSealFlattenersFB_BagFeed();
	msfVerticalAxis : FB_ThreePositionCylinder();
    pressureBar : FB_MotorizedPressureBar();
	IBD : FB_MotorizedIBD();
	sealBarTempSensor : FB_IFMTempSensor();
	sealBarHeater : FB_TempController();
    startCycleONS : R_TRIG;
	enableBagOpen : BOOL;
	enableLoadPlate : BOOL;
	enableHeater : BOOL;
	enableIBDDeflate : BOOL;
	enableIBDEject : BOOL;
	enableLabelSideUp : BOOL := TRUE;
	factoryTestModeKeepCycling : BOOL;
	autoModeKeepCycling : BOOL;
	autoModeKeepCyclingTimer : Standard.TON;
    bagDelivery : BagDeliveryFB();
    //zebraPrinter : PrinterFB;            //Printer Test Rig
	zebraPrinter : PrinterFB_Mode2;
	sealTimer : Standard.TON() := (PT := T#350MS);
	bagOpenFingerDelay : Standard.TON := (PT := T#100MS);
	bagDropTimer : Standard.TON;
	HPA : MonostableMultivibratorFB();
    rearLoadPlateRetract : MonostableMultivibratorFB() := (Dwellsetting := 1500);
	forwardLoadPlateRetract : MonostableMultivibratorFB() := (Dwellsetting := 1500);
	loadShelfExtend : MonostableMultivibratorFB() := (Dwellsetting := 1500);
	exitConveyorRun : DelayDwellFB() := (Dwellsetting := 6000);
	externalExitConveyorRun : DelayDwellFB() := (Dwellsetting := 6000);
	
	//IBDCylinders : FB_ThreePositionCylinder();
	IBDExtendONS : FB_ONS();
	IBDRetractONS : FB_ONS();
	//IBDRetractToDeflate : MonostableMultivibratorFB();
	//IBDRetractToEject : MonostableMultivibratorFB();
	bagOpenFingers : BagOpenFingersWithSensorsFB();
	bagOpenCheckDelay : Standard.TON := (PT:= T#400MS); // Delay to check if bag open
	bagOpenRetrySetting : UINT;		// Number of times to retry opening bag
	bagOpenRetryCount : UINT;		// Count of current retry attempts
	bagOpenFeedNewBagSetting : UINT; // Number of new bags to try
	bagOpenFeedNewBagCount : UINT;	// Count of new bags tried in recovery
	bagOpened : BOOL;				// Bag was Opened flag
	recoveryModeActive : BOOL; 		// Recovery Mode Active
	startCycleReqFromPalmButtons : BOOL;
	startCycleReqFromPalmButtonsONS : FB_ONS();
	pressureBarMotor : FB_AppliedMotionStepServoEIPPassthrough();
	IBDMotor : FB_AppliedMotionStepServoEIPPassthrough();
	jawClamps : FB_ThreePositionCylinder();
	//passthrough : AdjustablePassthroughFB();
	homeJawPB : BOOL;
    setPassthroughPB : BOOL;
	vacuumHoldTimer : Standard.TON() := (PT := T#250MS);
	cycleTimer : TON() := (PT := T#1000S);
	cycleTime : REAL;
	bagFailedToOpen : FB_Fault(name := 'Bag Failed to Open');
	openedBagWasRemoved : FB_Fault(name := 'Opened Bag was Removed');
	safePowerFailure : FB_Fault(name := 'E-Stop/Safety Power Failure');
	palmButtonConfigError : FB_Fault(name := 'Palm Button Configuration Error');
	packageEjectGuardRemoved : FB_Fault(name := 'Package Eject Guard Removed');
	barcodeVerificationFailed : FB_Fault(name := 'Barcode Verification Failed');
	barcodeVerifierCommFail : FB_Fault(name := 'Barcode Verifier Communication Failure');
	infeedConveyorIOCommFail : FB_Fault(name := 'Infeed Conveyor IO Communication Failure');
	infeedConveyorVFDFaulted : FB_Fault(name := 'Infeed Conveyor VFD Failure');
	printAndApplyFaulted : FB_Fault(name := 'Print and Apply Faulted');
	productJammed : FB_Fault(name := 'Product Jammed on Exit Conveyor');
	printAndApplyCommFailure : FB_Fault(name := 'Print and Apply Comm Failure');
	printAndApplyWaitForLabelTimedOut : FB_Fault(name := 'Print and Apply Timed Out');
	iPowerOffButtonONS : FB_ONS();
	loadPlateFaultTimer : FB_CylinderFaults();
	loadPlateFaults : LoadPlateFaultsType;
	forwardLoadPlateFaultTimer : FB_CylinderFaults();
	forwardLoadPlateFaults : LoadPlateFaultsType;
	rearLoadPlateFaultTimer : FB_CylinderFaults();
	rearLoadPlateFaults : LoadPlateFaultsType;
	loadShelfFaultTimer : FB_CylinderFaults();
	loadShelfFaults : LoadPlateFaultsType;
	LPA : DelayDwellFB();
	hpaServiceOnONS : FB_ONS;
	exitConveyorJogONS : FB_ONS;
	externalExitConveyorJogONS : FB_ONS;
	obstructionFaultONS : FB_ONS;
	hmiLight  : FB_HMILight;
	faultONS : FB_ONS;
	powerSettlingTimer : Standard.TON := (PT := T#6S);
	pressureBarCloseDelay : Standard.TON;
	filler : FillerFB();
	configOutput1Pulse : MonostableMultivibratorFB();
	configOutput2Pulse : MonostableMultivibratorFB();
	fillerModeCycleStartOnlyPulse : MonostableMultivibratorFB();
	murrIOBusNode : MurrIOFB();
	funnel : FunnelFB();
	barcodeVerifier : BarcodeReaderFB();
	keyenceBCV : KeyenceNL20FB();
	rearMotorCommsReturned : Standard.F_TRIG();
	baggerHeadMovement : FB_BaggerHeadRaise();
	resettingActive : BOOL;
	resetTimer : Standard.TOF := (PT := T#1S);
	allMotorCommsGood : BOOL;
	lightedPalmButton : FB_MurrK50;
	footSwitchONS : FB_ONS;
	IBDOutSetting: REAL;
	ezfeed : EZFeedFB();
	printAndApply : PrintAndApplyFB();
	EIPReconfig : FB_EIPCommsConfigure();
END_VAR

//    Function Block: FB_MOABHead
//    Description: This is the supervisory module for the MOAB head.
//    There is one supervisory state machine for the head and 3 sub-state machines Sealing/Separating, Release/Feed, and Opening Bag
//    Created by: Ben Hess
//    Created Date: Tuesday, April 17, 2018

{region "Setup"}
// Run BaseComponentFB
SUPER^();

EIPReconfig(rootEIPNode := EtherNet_IP_Scanner);
//EIPReconfig(rootEIPNode := Dual_LAN_Card);

// When power is returned, give machine ~5 seconds
powerSettlingTimer(IN := iEStopOK);
Globals.machinePowerOK := powerSettlingTimer.Q;
safePowerFailure.faultTrigger := NOT iEStopOK AND murrIOBusNode.ok;

// Bags Low warning
HMIData.bagLevelLow.active := iBagsLow;

// Ethernet/IP barcode verifier from Keyence
keyenceBCV(
	enable:= , 
	ptrEIPInputs:= ADR(keyenceBCVInputs), 
	ptrEIPOutputs:= ADR(keyenceBCVOutputs), 
	triggerInput:= , 
	lastReadData => HMIData.barcodeLastReadString);	 
// Barcode Verifier interface to printer
barcodeVerifier(enable := (HMIData.barcodeVerifierSelection <> BCVSelection.NotInstalled AND HMIData.barcodeVerifierInUse),
		 		readGoodInput := keyenceBCV.goodRead,
				distanceToScan := HMIData.barcodeScanDistance,
				feedSpeed := TO_REAL(HMIData.printSpeed),
				positionOffset := HMIData.barcodeStartPosition,
				badReadFaultCountSetting := HMIData.barcodeBadReadFaultSetting,
				currentBadReadCount => HMIData.barcodeBadReadCount,
				currentGoodReadCount => HMIData.barcodeGoodReadCount,
				triggerScannerOutput => keyenceBCV.triggerInput);
// Enable comms to Keyence N-L20 if selected in factory config
IF HMIData.barcodeVerifierSelection = BCVSelection.LaserScanner THEN
	Keyence_BCV.Enable := TRUE; 

	IF Keyence_BCV.eState <> IoDrvEthernetIP.AdapterState.RUNNING THEN 
		barcodeVerifierCommFail.Trigger();
	END_IF

ELSE
	Keyence_BCV.Enable := FALSE;
END_IF

// Raise/Lower bagger head logic
// Indications and commands from HMI
HMIData.baggerHeadService.extendedFeedback := NOT iHeadRaised;
HMIData.baggerHeadService.retractedFeedback := NOT iHeadLowered;
IF HMIData.baggerHeadService.retractedFeedback THEN
	HMIData.baggerHeadService.retractCommand := FALSE;
END_IF
IF HMIData.baggerHeadService.extendedFeedback THEN
	HMIData.baggerHeadService.extendCommand := FALSE;
END_IF
baggerHeadMovement(
	faultIndication:= HMIData.faultActive, 
	raiseCommand:= HMIData.baggerHeadService.extendCommand, 
	lowerCommand:= HMIData.baggerHeadService.retractCommand, 
	raiseLimitSwitch:= HMIData.baggerHeadService.extendedFeedback, 
	lowerLimitSwitch:= HMIData.baggerHeadService.retractedFeedback, 
	runMotorOutput=> oRunBaggerHeadMotor, 
	motorDirectionOutput=> oBaggerHeadMotorDir);
	 
// Option setup and factory config  
	 
IF HMIData.resetAverageCycleTime THEN
	HMIData.averageCycleTime := 0;
	HMIData.resetAverageCycleTime := FALSE;
END_IF
HMIData.lastCycleTime := cycleTime;

HMIData.printerNotReady.active := (NOT printerReady AND zebraPrinter.enable) OR (printAndApply.printerNotReady AND printAndApply.enable);
HMIData.waitingForPrinter.active := (zebraPrinter.state = PRINTER_STATES.WaitingForData AND releaseAndFeedSubState = RELEASE_FEED_STATES.WaitForPrinter) OR (printAndApply.waitingForPrinter AND printAndApply.enable);
//HMIData.printerRibbonLow.active := printerRibbonLow;
	 
batchSetting := HMIData.batchSetting;
HMIData.batchCount := batchCount;

bagOpenRetrySetting := HMIData.bagOpenRetrySetting;
HMIData.bagOpenRetryCount := bagOpenRetryCount;
	 
// Run bus node		  
murrIOBusNode(
	enable:= , 
	headNodeEnabled:= TRUE, 
	guardNodeEnabled:= (HMIData.cycleStartButtonSelection = PalmButtonSelection.SinglePalmButton 
						OR HMIData.cycleStartButtonSelection = PalmButtonSelection.DualPalmButton
						OR (HMIData.funnelFactorySelection <> FunnelSelection.NotInstalled)), 
	printerNodeEnabled:= , 
	dischargeNodeEnabled:= TRUE, 
	auxIONodeEnabled:= , 
	configVersion:= HMIData.murrIOConfigVersion, 
	ptrMachineOptionsManagementOutputs:= ADR(oMOMConfig), 
	ptrSystemStatusInputs:= ADR(iMurrSystemState));

// Setup of Motorized seal flattener motor and function block
msfVerticalAxis(extendOutput => oSealFlatDown, retractOutput => oSealFlatUp);
msfVerticalAxis.Execute();
motorizedSealFlatteners(sealFlattenersVerticalAxis := msfVerticalAxis,
						jogIn := HMIData.sealFlattenersServiceJogIn,
						jogOut := HMIData.sealFlattenersServiceJogOut,
						raiseService := HMIData.sealFlattenersServiceRaise,
						lowerService := HMIData.sealFlattenersServiceLower,
						moveToManualSetpoint := HMIData.sealFlattenersMoveToManualPos,
						manualPosSetpoint := HMIData.sealFlattenersManualPositionSetting,
						sealFlattenerMotorCommFailInput := MSFMotor.eState <> IoDrvEthernetIP.AdapterState.RUNNING);
motorizedSealFlatteners.Mode := motorizedSealFlattenersMode;
pressureBarMotor(ptrEIPInputs := ADR(jawPasstrhoughMotorInputs),
                ptrEIPOutputs := ADR(jawPasstrhoughMotorOutputs),
                stepsPerInchSetpoint := Globals.STEPS_PER_INCH_TFBelt,
                //faultHandler := PRG_Bagger.faultHandler,
				reversePolarity := FALSE,
				defaultCurrentSetpoint := 500,
				commFail := Pbar_ServoEIP.eState <> IoDrvEthernetIP.AdapterState.RUNNING,
				isHomable := TRUE);			
pressureBarMotor.Execute();

jawClamps(
	mode:= , 
	extendedStatus=> , 
	retractedStatus=> , 
	extendOutput=> oJawClampExtend, 
	retractOutput=> oJawClampRetract);	 
	 
pressureBar(
	enable:= , 
	iPressureBarClamped:= iJawClamped, 
	iPressureBarClosed:= iJawClearToClamp, 
	iPressureBarNotObstructed:= TRUE, 
	iBaggerEnableButton:= , 
	iJawClampExtended:= iJawClampsExtended, 
	iJawCLampRetracted:= iJawClampsRetracted, 
	pbarOutSetting:= HMIData.passthroughSetting, 
	pbarInSetting:= , 
	disableFaults:= , 
	extendJawClamp:= , 
	retractJawClamp:= , 
	extendJaw:= , 
	retractJaw:= , 
	faults => , 
	failToClampLeft=> , 
	failToReleaseLeft=> , 
	failToClampRight=> , 
	failToReleaseRight=> , 
	state=> , 
	actualPosition=> HMIData.passthroughPosition,
	pressureBarClosed => HMIData.pressureBarService.retractedFeedback,
	pressureBarOpen => HMIData.pressureBarService.extendedFeedback, 
	jawClamps:= jawClamps, 
	pbarMotor:= pressureBarMotor);
pressureBar.Mode := electricPressureBarMode;


// Run bag delivery 
bagDelivery(jogForwardPB := HMIData.jogBagForward,
			jogReversePB := HMIData.jogBagReverse,
			bagFeedMasterMotorCommFailInput := Bag_Delivery_EIP_Motor.eState <> IoDrvEthernetIP.AdapterState.RUNNING,
			bagFeedRearMotorCommFailInput := Bag_Delivery_Rear_Motor.eState <> IoDrvEthernetIP.AdapterState.RUNNING,
			stepsPerInchSetting := Globals.STEPS_PER_INCH_PRO24_BAG_DELIVERY);
bagDelivery.Mode := bagDeliveryMode;

CASE HMIData.baggerModelSelection OF
	ModelSelection.Pro18:
	
	ModelSelection.Pro18_02:
		 
	ModelSelection.Pro24:
END_CASE
	 
CASE HMIData.printerSelection OF
		 
	LabelPrinterSelection.NotInstalled:				//
													zebraPrinter.enable := FALSE;
													printAndApply.enable := FALSE;
													Panther_PA.Enable := FALSE;
													murrIOBusNode.printerNodeEnabled := FALSE;
	
	LabelPrinterSelection.ZebraPrinter203DPI, 			   
		LabelPrinterSelection.ZebraPrinter300DPI:	//
													zebraPrinter.enable := HMIData.printerInUse;
													printAndApply.enable := FALSE;
													Panther_PA.Enable := FALSE;
													murrIOBusNode.printerNodeEnabled := TRUE;
														 
			
	LabelPrinterSelection.PrintAndApply203DPI,
		LabelPrinterSelection.PrintAndApply300DPI:			//
		 											zebraPrinter.enable := FALSE;
													Panther_PA.Enable := TRUE;
													printAndApply.enable := HMIData.printerInUse;
													murrIOBusNode.printerNodeEnabled := FALSE;
END_CASE



	 
// Run Zebra Printer
zebraPrinter(ribbonEncoderPulse := iPrinterRibbonEncoder, oLowerPrintHead => oPrintHeadDown);
zebraPrinter.Mode := printerMode;
IF HMIData.activateDemoMode THEN
	HMIData.demoModeIsActive.active := TRUE;
	zebraPrinter.autoSendLabel := TRUE;
ELSE
	HMIData.demoModeIsActive.active := FALSE;
	zebraPrinter.autoSendLabel := FALSE;
END_IF

printAndApply(
	enable:= , 
	bypass := NOT bagOpened,
	baggerFaulted:= HMIData.faultActive, 
	baggerInCycle:= HMIData.inCycle, 
	dataReady:= iPAOnlineDataReady, 
	LOTAR:= iPALOTAR, 
	faultInput:= NOT iPAFaulted,
	PACycleComplete:= iPACycleComplete, 
	applicatorHome:= iPAApplicatorHome, 
	heartbeat:= iPAHeartbeat, 
	productSensor:= NOT iConveyorClear, 
	exitConveyorRunAfterPASetting := HMIData.printAndApplyConveyorDwell,
	waitForPrinterFaultSetting := HMIData.printAndApplyWaitForLabelTimeout,
	state=> , 
	commFail=> printAndApplyCommFailure.faultTrigger, 
	faultedStatus=> printAndApplyFaulted.faultTrigger, 
	waitForPrintFault=> printAndApplyWaitForLabelTimedOut.faultTrigger,
	printerNotReady=> , 
	printerReadyToApply=> , 
	waitingForPrinter=> , 
	triggerOutput=> oPATrigger1,
	resetOutput=> oPAReset, 
	inhibitCycle=> , 
	inhibitConveyor=> );
	 
// Run funnel
funnel(
	enable:= HMIData.funnelFactorySelection <> FunnelSelection.NotInstalled AND HMIData.funnelInUse, 
	sensorsInstalled:= HMIData.funnelFactorySelection = FunnelSelection.FunnelWithSensors, 
	openSensor:= iFunnelOpened, 
	closedSensor:= iFunnelClosed, 
	opened=> , 
	closed=> , 
	closeOutput=> oIBDRetract, 
	openOutput=> oIBDExtend, 
	failToOpen=> , 
	failToClose=> );
funnel.OpeningTime := HMIData.funnelOpeningTime;
funnel.ClosingTime := HMIData.funnelClosingTime;
funnel.DelaySetting := HMIData.funnelOpenDelay;
// Setup of pick and place motors


sealBarTempSensor(ptrTemperatureBytes := ADR(iHeaterBarTempInputs));
sealBarTempSensor.Execute();
sealBarHeater(enable := NOT safePowerFailure.active,
				temperatureSensor := sealBarTempSensor,
				temperatureSetpoint := TO_REAL(HMIData.sealBarTemperatureSetting),
				heaterPulse => 	oHeaterPulse);	  
HMIData.sealBarTemperature := TO_UDINT(sealBarHeater.currentTemp);
{region "timers"}
// Timers
sealTimer();
bagOpenFingerDelay();
vacuumHoldTimer(PT := TO_TIME(HMIData.vacuumDwell * 1000));
bagOpenCheckDelay();
bagDropTimer(PT := TO_TIME((HMIData.loadPlateDelay * 1000) + (HMIData.bagDropTime * 1000)));
{endregion}
		  
// Setup of HPA and load plate.  Use .Trigger() to run.
HPA.DwellSetting := TO_UINT(HMIData.hpaDwell * 1000);
HPA(Q => oHPAOn);
hpaServiceOnONS(CLK := HMIData.hpaserviceOn);

LPA.DwellSetting := TO_DINT(HMIData.lpaDwell * 1000);
LPA(Q => oLPAOn);
	 
CASE HMIData.independentBagDeflatorSelection OF
	BagDeflatorSelection.NotInstalled:					// Disable IBD
		 													enableIBDDeflate := FALSE;
															enableIBDEject := FALSE;
	
	BagDeflatorSelection.IBDStandard:	// Enable IBD
															IF HMIData.IBDDeflateDwellTime <> 0 THEN
																enableIBDDeflate := TRUE;
															ELSE
																enableIBDDeflate := FALSE;
															END_IF
															
															IF HMIData.IBDPackageEjectAssistDwellTime <> 0 THEN
																enableIBDEject := TRUE;
															ELSE
																enableIBDEject := FALSE;
															END_IF
	 														
																 
	BagDeflatorSelection.IBDWithHingedPlate:	// Enable IBD with Hinged Plate
															
																 
	BagDeflatorSelection.MotorizedIBD:			// Enable motorized IBD
															IF HMIData.IBDDeflateDwellTime <> 0 THEN
																enableIBDDeflate := TRUE;
															ELSE
																enableIBDDeflate := FALSE;
															END_IF
															
															IF HMIData.IBDPackageEjectAssistDwellTime <> 0 THEN
																enableIBDEject := TRUE;
															ELSE
																enableIBDEject := FALSE;
															END_IF
	
END_CASE

CASE HMIData.bofSelection OF
	BagOpenFingersSelection.NotInstalled:					// Disable Bag Open
		 													enableBagOpen := FALSE;
															
	
	BagOpenFingersSelection.PneumaticWithBagOpenSensors:	// Enable Bag Open
															enableBagOpen := TRUE;
	
END_CASE


CASE HMIData.packageEjectSelection OF
	PackageEjectionSelection.NotInstalled:				// Disable all
														enableLoadPlate := FALSE;
														enableLabelSideUp := FALSE;	
														loadPlateFaultTimer.enable := FALSE;	
														forwardLoadPlateFaultTimer.enable := FALSE;
														rearLoadPlateFaultTimer.enable := FALSE;
														loadShelfFaultTimer.enable := FALSE;
		 
	PackageEjectionSelection.RearRetractingLoadPlate:	// Enable rear retracting load plate
		 												enableLoadPlate := TRUE;
														enableLabelSideUp := FALSE;	
														loadPlateFaultTimer.enable := Globals.machinePowerOK;	
														forwardLoadPlateFaultTimer.enable := FALSE;
														rearLoadPlateFaultTimer.enable := FALSE;
														loadShelfFaultTimer.enable := FALSE;
														rearLoadPlateRetract.DelaySetting := TO_UINT(HMIData.loadPlateDelay * 1000);
														rearLoadPlateRetract.DwellSetting := TO_UINT(HMIData.loadPlateDwell * 1000);
	
	PackageEjectionSelection.LabelSideUp:				// Enable all
		 												enableLoadPlate := TRUE;
														enableLabelSideUp := TRUE;	
														loadPlateFaultTimer.enable := FALSE;
														forwardLoadPlateFaultTimer.enable := (state >= HEAD_STATES.ReleaseAndFeedBag) AND HMIData.inCycle;
														rearLoadPlateFaultTimer.enable := Globals.machinePowerOK;
														//loadShelfFaultTimer.enable := Globals.machinePowerOK;
														rearLoadPlateRetract.DelaySetting := 0;
														rearLoadPlateRetract.DwellSetting := TO_UINT((HMIData.loadPlateDwell + HMIData.loadPlateDelay) * 1000);
END_CASE

CASE HMIData.cycleStartButtonSelection OF
	PalmButtonSelection.NotInstalled:					// Dont' allow input to start bagger cycle
		 												startCycleReqFromPalmButtons := FALSE;
		 
	PalmButtonSelection.SinglePalmButton:				// Start using one side only
		 												startCycleReqFromPalmButtons := iRightPalmButton;
														
														// Trigger fault if left palm button is seen - should be set up for dual!	 
														IF iLeftPalmButton THEN
															palmButtonConfigError.Trigger();		 
														END_IF
		 
	PalmButtonSelection.DualPalmButton:					// Both buttons must be pressed
		 												startCycleReqFromPalmButtons := iRightPalmButton AND iLeftPalmButton;
															 
	PalmButtonSelection.LightedPalmButton:				// Lighted Murr palm button input comes from IO Link
		 												startCycleReqFromPalmButtons := iMurrTouchButtonStatus.0;
															 
END_CASE
startCycleReqFromPalmButtonsONS(CLK := startCycleReqFromPalmButtons);	 

lightedPalmButton(	baggerReady:= readyToRun AND NOT HMIData.sealBarNotAtTemperature.active, 
					baggerFaulted:= HMIData.faultActive, 
					baggerInCycle:= HMIData.inCycle, 
					IOLinkStateOutput=> oMurrTouchbuttonState);

		  
CASE HMIData.auxIOConfig.factorySelection OF
	AuxiliaryIOSelection.NotInstalled:					// Turn outputs off
		 												oAuxBaggerOK := FALSE;
														oAuxReadyForFiller := FALSE;
														configOutput1Pulse.ManualOff();	
														configOutput1Pulse.Reset();
														configOutput2Pulse.ManualOff();	
														configOutput2Pulse.Reset();
														murrIOBusNode.auxIONodeEnabled := FALSE;
														HMIData.fillerFactorySelection := FillerSelection.NotInstalled;
		 
	AuxiliaryIOSelection.AuxIOStandard:					// Use aux IO
		 												murrIOBusNode.auxIONodeEnabled := TRUE;
		 												oAuxBaggerOK := NOT HMIData.faultActive;
														oAuxReadyForFiller := filler.waitingForFiller;
															 
 														CASE HMIData.auxIOConfig.cfgInputSelection OF
															AuxInputSelection.NotConfigured:		// 
																									HMIData.baggerInhibited.active := printAndApply.inhibitCycle;
																										 
															AuxInputSelection.BaggerInhibit:		//
																 									HMIData.baggerInhibited.active := iAuxConfigInput OR printAndApply.inhibitCycle;
														END_CASE
 
														CASE HMIData.auxIOConfig.cfgOutput1Selection OF
																 
															AuxOutputSelection.BagMade:				//
																 									IF state = HEAD_STATES.SealedAndSeparatedBag THEN
																										configOutput1Pulse.Trigger();
																									END_IF
																										 
															AuxOutputSelection.CycleComplete:		//
																 									IF state = HEAD_STATES.OpenedBag THEN
																										configOutput1Pulse.Trigger();
																									END_IF
																										 
															AuxOutputSelection.PrinterDataReady:	//
																 									IF printerDataReady THEN
																										configOutput1Pulse.ManualOn();
																									ELSE
																										configOutput1Pulse.ManualOff();
																									END_IF
																										 
															AuxOutputSelection.WaitingForPrinter:	// 
																 									IF releaseAndFeedSubState = RELEASE_FEED_STATES.WaitForPrinter THEN
																										configOutput1Pulse.ManualOn();
																									ELSE
																										configOutput1Pulse.ManualOff();	
																								    END_IF
																										 
															AuxOutputSelection.BagMadePlusLabelRequired:	//
																 									IF NOT printerDataReady AND state = HEAD_STATES.SealedAndSeparatedBag THEN
																										configOutput1Pulse.ManualOn();
																									END_IF
																									
																									IF printerDataReady OR HMIData.faultActive OR (releaseAndFeedSubState = RELEASE_FEED_STATES.FeedToOffset) THEN
																										configOutput1Pulse.ManualOff();
																									END_IF 
															AuxOutputSelection.BagsLow:				//
																									IF HMIData.bagLevelLow.active THEN
																										configOutput1Pulse.ManualOn();
																									ELSE
																										configOutput1Pulse.ManualOff();
																									END_IF											 
															
														END_CASE
															 
														CASE HMIData.auxIOConfig.cfgOutput2Selection OF
																 
															AuxOutputSelection.BagMade:				//
																 									IF state = HEAD_STATES.SealedAndSeparatedBag THEN
																										configOutput2Pulse.Trigger();
																									END_IF
																										 
															AuxOutputSelection.CycleComplete:		//
																 									IF state = HEAD_STATES.OpenedBag THEN
																										configOutput2Pulse.Trigger();
																									END_IF
																										 
															AuxOutputSelection.PrinterDataReady:	//
																 									IF printerDataReady THEN
																										configOutput2Pulse.ManualOn();
																									ELSE
																										configOutput2Pulse.ManualOff();
																									END_IF
																										 
															AuxOutputSelection.WaitingForPrinter:	// 
																 									IF releaseAndFeedSubState = RELEASE_FEED_STATES.WaitForPrinter THEN
																										configOutput2Pulse.ManualOn();
																									ELSE
																										configOutput2Pulse.ManualOff();	
																								    END_IF
																										 
															AuxOutputSelection.BagMadePlusLabelRequired:	//
																 									IF NOT printerDataReady AND state = HEAD_STATES.SealedAndSeparatedBag THEN
																										configOutput2Pulse.ManualOn();
																									END_IF
																									
																									IF printerDataReady OR HMIData.faultActive OR (releaseAndFeedSubState = RELEASE_FEED_STATES.FeedToOffset) THEN
																										configOutput2Pulse.ManualOff();
																									END_IF 
																										 
															AuxOutputSelection.BagsLow:				//
																									IF HMIData.bagLevelLow.active THEN
																										configOutput2Pulse.ManualOn();
																									ELSE
																										configOutput2Pulse.ManualOff();
																									END_IF	
														END_CASE
														
		 
END_CASE 
	 
// Pulse outputs that are temporary statuses (Cycle Complete) vs. held (Waiting for Printer) 
configOutput1Pulse(Q => oAuxConfigOut1);
configOutput2Pulse(Q => oAuxConfigOut2);
configOutput1Pulse.DwellSetting := 500;
configOutput2Pulse.DwellSetting := 500;

// Filler and EZFeed conveyor setup
CASE HMIData.fillerFactorySelection OF
	FillerSelection.NotInstalled:					// No filler
		 											filler.enable := FALSE;
													filler.activateFiller := FALSE;	
													ezfeed.enable := FALSE;
													fillerModeCycleStartOnlyPulse.Reset();
													Infeed_Conveyor_IO.Enable := FALSE;
		 
	FillerSelection.StandardFiller:					// Only enable filler if Aux IO is enabled
		 											filler.enable := (HMIData.auxIOConfig.factorySelection = AuxiliaryIOSelection.AuxIOStandard);
													Infeed_Conveyor_IO.Enable := FALSE;
														 
	FillerSelection.EZFeed:							filler.enable := TRUE;
		 											ezfeed.enable := TRUE;
													Infeed_Conveyor_IO.Enable := TRUE;
													
		 											

END_CASE 	 

ezfeed(
	enable:= , 
	baggerFaulted:= HMIData.faultActive, 
	enableEZFeed:= HMIData.fillerEnable, 
	continuousModeEnable:= HMIData.infeedConveyorRunningMode, 
	partsCountingModeEnable:= HMIData.infeedConveyorCountingMode, 
	flightPresentSensor:= iInfeedFlightSensor, 
	partPresentSensor:= , 
	waitingForFiller:= filler.waitingForFiller, 
	indexDwellSetting:= HMIData.infeedIndexDwellTimer, 
	flightTarget:= HMIData.infeedFlightCountTarget, 
	partsTarget:= HMIData.infeedPartsCountTarget, 
	emptyPartsWarningSetting:= HMIData.infeedEmptyPartsSetting, 
	restartFromEmptyParts:= HMIData.initiateCycle, 
	state=> , 
	runVFD=> oRunInfeedVFD, 
	flightCount=> HMIData.infeedFlightCountActual, 
	partsCount=> HMIData.infeedPartsCountActual, 
	emptyPartsWarningCount=> HMIData.infeedEmptyPartsActual, 
	emptyPartsWarning=> HMIData.infeedConveyorOutOfParts.active,
	EZFeedDone=> );

IF HMIData.fillerFactorySelection = FillerSelection.EZFeed THEN
	Infeed_Conveyor_IO.Enable := TRUE; 

	IF Infeed_Conveyor_IO.eState <> IoDrvEthernetIP.AdapterState.RUNNING THEN 
		infeedConveyorIOCommFail.Trigger();
	END_IF
ELSE
	Infeed_Conveyor_IO.Enable := FALSE;
END_IF
	 
infeedConveyorVFDFaulted.faultTrigger := (HMIData.fillerFactorySelection = FillerSelection.EZFeed) AND NOT iInfeedVFDNotFaulted;
		 
fillerModeCycleStartOnlyPulse.DwellSetting := 4000;
fillerModeCycleStartOnlyPulse(Q => HMIData.fillerModeCycleStartOnly.active);
filler(
	enable:= , 
	fillerTrigger:= iAuxFillerTrigger OR ezfeed.EZFeedDone,
	fillerOK:= iAuxFillerOK, 
	activateFiller:= HMIData.fillerEnable, 
	dropTime:= HMIData.fillerDropTime,
	state=> , 
	fillerModeActive=> , 
	waitingForFiller=> ,
	cycleBagRequest=> , 
	cycleBaggerToActivateFiller=> , 
	notReady=> );	 
IF filler.activateFiller AND NOT filler.cycleBaggerToActivateFiller.active THEN
	IF HMIData.initiateCycle OR startCycleReqFromPalmButtons THEN
		fillerModeCycleStartOnlyPulse.Trigger();
	END_IF
END_IF
	 

//HMIData.packageEjectGuardRemoved.active :=  HMIData.packageEjectSelection = PackageEjectionSelection.LabelSideUp AND NOT iPackageEjectGuardClosed;
HMIData.loadPlateService.extendedFeedback := HMIData.rearLoadPlateService.extendedFeedback := iLoadPlateExtended;
HMIData.loadPlateService.retractedFeedback := HMIData.rearLoadPlateService.retractedFeedback := iLoadPlateRetracted;

rearLoadPlateRetract();
oLoadPlateRetract := rearLoadPlateRetract.Q;
oLoadPlateExtend := NOT oLoadPlateRetract;
loadPlateFaultTimer(
	enable:= , 
	extendCommand:= oLoadPlateExtend, 
	extendedInput:= iLoadPlateExtended, 
	retractCommand:= oLoadPlateRetract, 
	retractedInput:= iLoadPlateRetracted, 
	faultTime:= , 
	failToExtend=> loadPlateFaults.failedToLoad.faultTrigger, 
	failToRetract=> loadPlateFaults.failedToDischarge.faultTrigger);
rearLoadPlateFaultTimer(
	enable:= , 
	extendCommand:= oLoadPlateExtend, 
	extendedInput:= iLoadPlateExtended, 
	retractCommand:= oLoadPlateRetract, 
	retractedInput:= iLoadPlateRetracted, 
	faultTime:= , 
	failToExtend=> rearLoadPlateFaults.failedToLoad.faultTrigger, 
	failToRetract=> rearLoadPlateFaults.failedToDischarge.faultTrigger);

HMIData.forwardLoadPlateService.extendedFeedback := iFrontLoadPlateExtended;
HMIData.forwardLoadPlateService.retractedFeedback := iFrontLoadPlateRetracted;
forwardLoadPlateRetract.DwellSetting := TO_UINT(HMIData.loadPlateDwell * 1000);
forwardLoadPlateRetract.DelaySetting := TO_UINT(HMIData.loadPlateDelay * 1000);
forwardLoadPlateRetract();
oFrontLoadPlateToLoad := NOT forwardLoadPlateRetract.Q;
oFrontLoadPlateToDischarge := NOT oFrontLoadPlateToLoad;
forwardLoadPlateFaultTimer(
	enable:= , 
	extendCommand:= NOT oFrontLoadPlateToLoad, 
	extendedInput:=iFrontLoadPlateExtended, 
	retractCommand:= oFrontLoadPlateToLoad, 
	retractedInput:= iFrontLoadPlateRetracted, 
	faultTime:= , 
	failToExtend=> forwardLoadPlateFaults.failedToLoad.faultTrigger, 
	failToRetract=> forwardLoadPlateFaults.failedToDischarge.faultTrigger);
		 
HMIData.loadShelfService.extendedFeedback := iLoadShelfExtended;
HMIData.loadShelfService.retractedFeedback := iLoadShelfRetracted;
loadShelfExtend.DwellSetting := TO_UINT(HMIData.loadPlateDwell * 1000);
loadShelfExtend.DelaySetting := TO_UINT(HMIData.loadPlateDelay * 1000);
loadShelfExtend();
oLoadShelfUp := NOT loadShelfExtend.Q;
loadShelfFaultTimer(
	enable:= , 
	extendCommand:= NOT oLoadShelfUp, 
	extendedInput:=iLoadShelfExtended, 
	retractCommand:= oLoadShelfUp, 
	retractedInput:= iLoadShelfRetracted, 
	faultTime:= , 
	failToExtend=> loadShelfFaults.failedToDischarge.faultTrigger, 
	failToRetract=> loadShelfFaults.failedToLoad.faultTrigger);
 
exitConveyorRun();
exitConveyorRun.DwellSetting := TO_DINT(HMIData.exitConveyorDwell * 1000);
exitConveyorJogONS(CLK := HMIData.exitConveyorJog);

IF printAndApply.inhibitConveyor THEN
	exitConveyorRun.Reset();
	externalExitConveyorRun.Reset();
END_IF


	 
oRunExitConveyor := ((exitConveyorRun.Q OR printAndApply.runConveyorAfterApply) AND HMIData.integratedExitConveyorSelection = IntegratedConveyorSelection.RearExit);
	 
externalExitConveyorRun();
externalExitConveyorRun.DwellSetting := TO_UINT(HMIData.externalExitConveyorDwell * 1000);
externalExitConveyorJogONS(CLK := HMIData.externalExitConveyorJog);
oRunExternalExitConveyor := ((externalExitConveyorRun.Q OR printAndApply.runConveyorAfterApply) AND HMIData.externalExitConveyorSelection <> ExteralConveyorSelection.NotInstalled);

bagOpenFingers(enable := HMIData.bofSelection <> BagOpenFingersSelection.NotInstalled,
				releaseOutput => oBOFUp,
		 		grabOutput => oBOFDown,
				rightFingerBagPresent := iRightFingerBagPresent,
				leftFingerBagPreset := iLefttFingerBagPresent,
				bagFailedToGrabBothFingersCount := Globals.bagFailedToGrabBothFingersCount,
				bagFailedToGrabLeftFingerCount := Globals.bagFailedToGrabLeftFingerCount,
				bagFailedToGrabRightFingerCount := Globals.bagFailedToGrabRightFingerCount,
				successfulBagOpenCount := Globals.successfulBagOpenCount);
					 


// Setup and run adjustable passthrough
//refIECObject := Pbar_ServoEIP;

	 
IBDMotor(ptrEIPInputs := ADR(iIBDMotorEIP),
                ptrEIPOutputs := ADR(oIBDMotorEIP),
                stepsPerInchSetpoint := Globals.STEPS_PER_INCH_TFBelt,
                //faultHandler := PRG_Bagger.faultHandler,
				reversePolarity := FALSE,
				defaultCurrentSetpoint := 650,
				//commFail := IBD_Motor.eState <> IoDrvEthernetIP.AdapterState.RUNNING,
				commFail := IBD_Motor.eState <> IoDrvEthernetIP.AdapterState.RUNNING,
				isHomable := TRUE);
IBDMotor.Execute();


IF HMIData.passthroughSetting + HMIData.IBDOffset > 12.0 THEN
	 IBDOutSetting := 12.0;
ELSE
	IBDOutSetting := HMIData.passthroughSetting + HMIData.IBDOffset;
END_IF
		  
IBD(
	enable:= , 
	pbarOutSetting:= IBDOutSetting, 
	pbarInSetting:= , 
	disableFaults:= , 
	extendCommand:= HMIData.IBDService.extendCommand, 
	retractCommand:= HMIData.IBDService.retractCommand ,  
	failToOpen=> , 
	state=> , 
	actualPosition=> , 
	IBDOpen=> , 
	homeRequired=> , 
	clamped=> , 
	IBDMotor:= IBDMotor);

obstructionFaultONS(CLK := (pressureBar.faults.obstructionDetected.active OR pressureBar.faults.failedToClose.active));
IF obstructionFaultONS.OSR THEN
	IBD.RemovePower();
END_IF
		 
IF HMIData.IBDService.extendCommand THEN
	HMIData.IBDService.extendCommand := FALSE;
END_IF
	 
IF HMIData.IBDService.retractCommand THEN
	HMIData.IBDService.retractCommand := FALSE;
END_IF
{endregion}
	 
hmiLight(lightOutput => oHMILight);
faultONS(CLK := HMIData.faultActive);

readyToRun := (motorizedSealFlatteners.Ready OR NOT motorizedSealFlatteners.enable) 
                AND (pressureBar.Ready OR NOT pressureBar.enable)
				AND (IBD.Ready OR NOT enableIBDDeflate)
                AND (bagDelivery.Ready OR NOT bagDelivery.enable)
                AND (zebraPrinter.Ready OR NOT zebraPrinter.enable)
				AND murrIOBusNode.ok;
iPowerOffButtonONS(CLK := iPowerOffButton);
resetTimer(IN := iPowerOffButtonONS.OSR);

allMotorCommsGood := NOT motorizedSealFlatteners.sealFlattenersHorizontalAxisMotor.faults.commFail.active
					AND NOT IBDMotor.faults.commFail.active
					AND NOT pressureBarMotor.faults.commFail.active
					AND NOT bagDelivery.bagfeedMasterMotor.faults.commFail.active
					AND NOT bagDelivery.bagFeedRearMotor.faults.commFail.active;

IF iPowerOffButtonONS.OSR THEN
	reset();
END_IF
			
IF HMIData.makeReady OR resetTimer.Q THEN
	Cube67_BN_E_V2.xAcknowledge := TRUE;
	FestoManifold.xAcknowledge := TRUE;
	MSFMotor.xAcknowledge := TRUE;
	Bag_Delivery_EIP_Motor.xAcknowledge := TRUE;
	Pbar_ServoEIP.xAcknowledge := TRUE;
	Bag_Delivery_Rear_Motor.xAcknowledge := TRUE;
	Keyence_BCV.xAcknowledge := TRUE;
	IBD_MOtor.xAcknowledge := TRUE;
	Panther_PA.xAcknowledge := TRUE;
	
	HMIData.ackAllFaults := TRUE;
	enable := TRUE;
	
	printAndApply.Reset();
	
	bagDropTimer.IN := FALSE;
	
	motorizedSealFlattenersMode := DEVICE_MODES.Auto;
	motorizedSealFlatteners.Reset();
	motorizedSealFlatteners.enable := HMIData.sealFlattenersSelection = SealFlattenerSelection.MotorizedSealFlatteners;
	
	HMIData.bagOpenFeedNewBagCount := 0;
	bagOpenRetryCount := 0;
	
	HMIData.stopMachine := FALSE;
	
	electricPressureBarMode := DEVICE_MODES.Auto;
	
	pressureBar.enable := TRUE;
	//pressureBar.ExtendCylinderLowPressure();
	
	//HMIData.sealBarTemperatureSetting := 300;
	enableHeater := TRUE;
	
	bagDeliveryMode := DEVICE_MODES.Auto;
	bagDelivery.Reset();
	bagDelivery.enable := TRUE;
	//bagDelivery.bagFeedMasterMotor.SetRearMotorToTorqueMode();
	IF iPowerOffButtonONS.OSR THEN
		bagDelivery.AutoFeedToEye();
	END_IF
	
	IF NOT bagOpenFingers.CheckIfBagGrabbed(FALSE) THEN
		bagOpened := FALSE;
	END_IF
	//bagOpened := FALSE;
	
	enableBatch := FALSE;
	batchCount := 0;
	
	//zebraPrinter.autoSendLabel := TRUE;
	printerMode := DEVICE_MODES.Auto;
	zebraPrinter.Reset();
	//zebraPrinter.enable := TRUE;
	
	IF iPowerOffButtonONS.OSR AND NOT bagDelivery.bagTensionFault.active THEN
		IF (HMIData.factoryTestMode AND (HMIData.bagsMade.count < 1000)) THEN
			HMIData.bagsMade.Clear();
		END_IF 
	END_IF  
	
	//passthrough.Reset();
	pressureBarMotor.Reset();
	passthroughMode := DEVICE_MODES.Auto;
	//passthrough.enable := TRUE;
	
	oVacOn := FALSE;
	rearLoadPlateRetract.Reset();
	forwardLoadPlateRetract.Reset();
	loadShelfExtend.Reset();
	
	LPA.Reset();
	LPA.ManualOff();
	HPA.Reset();
	funnel.CloseNow();
	exitConveyorRun.Reset();
	externalExitConveyorRun.Reset();
	oSealBarExtend := FALSE;
	oSealBarRetract := TRUE;
	sealTimer.IN := FALSE;
	pressureBarCloseDelay.IN := FALSE;
	filler.Reset();
	configOutput1Pulse.Reset();
	configOutput2Pulse.Reset();
	configOutput1Pulse.ManualOff();
	configOutput2Pulse.ManualOff();
	fillerModeCycleStartOnlyPulse.Reset();
	barcodeVerifier.Reset();
	keyenceBCV.Reset();
	state := HEAD_STATES.Idle;
	
	setPassthroughPB := FALSE;
	//homeJawPB := FALSE;
	HMIData.jobLoadRequired.active := TRUE;
	HMIData.makeReady := FALSE;
	bagDelivery.bagFeedRearMotor.SetRearMotorTorqueValue(TO_DINT(HMIDAta.bagTensionSetting * 100));
	hmiLight.TurnOff();
ELSE
	Cube67_BN_E_V2.xAcknowledge := FALSE;
	FestoManifold.xAcknowledge := FALSE;
	MSFMotor.xAcknowledge := FALSE;
	Bag_Delivery_EIP_Motor.xAcknowledge := FALSE;
	Pbar_ServoEIP.xAcknowledge := FALSE;
	Bag_Delivery_Rear_Motor.xAcknowledge := FALSE;
	Keyence_BCV.xAcknowledge := FALSE;
	IBD_MOtor.xAcknowledge := FALSE;
	Panther_PA.xAcknowledge := FALSE;
END_IF

IF enableONS.Q OR resetONS.Q THEN
    state := HEAD_STATES.Idle;
	sealAndSeparateSubState := SEAL_SEPARATE_STATES.Idle;
	releaseAndFeedSubState := RELEASE_FEED_STATES.Idle;
	openBagSubState := BAG_OPEN_ASSIST_STATES.Idle;
	finishCycleSubState := FINISH_CYCLE_STATES.Idle;
	motorizedSealFlatteners.Reset();
	pressureBar.Reset();
	IBD.Reset();
	bagDelivery.Reset();
	zebraPrinter.Reset();
	homeJawPB := FALSE;
	//EIPReconfig.ManualReconfig();
	IF IBD.homeRequired THEN
		homeJawPB := TRUE;
	ELSE
		//IBD.OpenIBD();
		homeJawPB := TRUE;
	END_IF
	IF pressureBar.homeRequired THEN
		homeJawPB := TRUE;
	ELSE
		//pressureBar.OpenJaw();
		homeJawPB := TRUE;
	END_IF
	//pressureBar.ExtendCylinderLowPressure();
	bagDropTimer.IN := FALSE;
	_reset := FALSE;
	cycleTimer.IN := FALSE;
//	bagFailedToOpen := FALSE;
END_IF

IF HMIData.bagsMade.count >= 1000 THEN
	Globals.factoryTestComplete := TRUE;
END_IF

IF Globals.factoryTestComplete THEN
	HMIData.machineNotTested.active := FALSE;
ELSE
	HMIData.machineNotTested.active := TRUE;
END_IF

IF HMIData.factoryTestMode THEN
	HMIData.factoryTestModeActive.active := TRUE;
ELSE
	HMIData.factoryTestModeActive.active := FALSE;
END_IF

// Disable the printer on dry cycle because we dont't want to print on the platen roller               
IF Globals.enableDryCycle THEN
    zebraPrinter.enable := FALSE;
END_IF

// Send torque value to motor                 
rearMotorCommsReturned(CLK := bagDelivery.bagFeedRearMotor.commFail);
IF HMIData.jobLoaded OR rearMotorCommsReturned.Q THEN
	bagDelivery.bagFeedRearMotor.SetRearMotorTorqueValue((TO_DINT(HMIData.bagTensionSetting * 100)));
END_IF

// Clear batch count on batch enable
enableBatchONS(CLK := enableBatch);
IF enableBatchONS.Q THEN
    batchCount := 0;
END_IF

//IF NOT enable OR NOT readyToRun OR faultONS.OSR THEN
IF NOT enable OR faultONS.OSR THEN
    state := HEAD_STATES.Fault;
	enableBatch := FALSE;
	//pressureBarMotor.Stop();
	cycleTimer.IN := FALSE;
END_IF
pressureBarCloseDelay(PT := TO_TIME(HMIData.pressureBarCloseDelay * 1000));
cycleTimer();
autoModeKeepCyclingTimer(PT := TO_TIME(HMIData.autoDwell * 1000), IN := autoModeKeepCycling AND state = HEAD_STATES.Idle);

HMIData.mayCycleUnexpectedly.active := autoModeSelected OR filler.activateFiller;

footSwitchONS(CLK := iFootSwitch);

IF state <> HEAD_STATES.Idle AND HMIData.initiateCycle THEN
	HMIData.initiateCycle := FALSE;
END_IF
CASE state OF
    HEAD_STATES.Idle :                                // Start cycle if enabled
													
													
                                                    IF (startCycle AND (filler.cycleBaggerToActivateFiller.active OR NOT filler.activateFiller)
													OR (enableBatch AND (batchCount < batchSetting))
													OR (HMIData.factoryTestMode AND (HMIData.bagsMade.count < 1000)) AND (factoryTestModeKeepCycling AND NOT LPA.Q)
													OR (startCycleReqFromPalmButtonsONS.OSR) AND (filler.cycleBaggerToActivateFiller.active OR NOT filler.activateFiller)
													OR (HMIData.initiateCycle AND readyToRun) AND (filler.cycleBaggerToActivateFiller.active OR NOT filler.activateFiller)
													OR (filler.cycleBagRequest AND HMIData.autoEnable)
													OR (filler.cycleBagRequest AND NOT HMIData.autoEnable) AND (footSwitchONS.OSR OR HMIData.initiateCycle OR startCycleReqFromPalmButtonsONS.OSR)
													OR (autoModeKeepCyclingTimer.Q)
													OR footSwitchONS.OSR)
													AND (NOT HMIData.faultActive 
													AND NOT HMIData.stopMachine 
													AND NOT HMIData.baggerInhibited.active
													AND NOT HMIData.sealBarNotAtTemperature.active
													AND NOT setPassthroughPB)
													AND readyToRun 
													THEN
                                                        state := HEAD_STATES.SealAndSeparateBag;
                                                        startCycle := FALSE;
														
														cycleTimer.IN := TRUE;
                                                    END_IF
													IF NOT Globals.passthroughChangedFromJog AND HMIData.jobLoaded THEN
														HMIData.jobLoaded := FALSE;
													END_IF
                                                    IF (HMIData.passthroughSetting <> passthroughSettingLast) OR (Globals.passthroughChangedFromJog AND HMIData.jobLoaded) AND NOT pressureBarMotor.Faulted AND NOT pressureBarMotor.HomeRequired THEN
															setPassthroughPB := TRUE;
															Globals.passthroughChangedFromJog := FALSE;
															HMIData.jobLoaded := FALSE;
															passthroughSetting := HMIData.passthroughSetting;
															passthroughSettingLast := HMIData.passthroughSetting;
													END_IF
													
													IF (NOT pressureBarMotor.HomeRequired OR pressureBarMotor.Faulted)
														AND (NOT motorizedSealFlatteners.sealFlattenersHorizontalAxisMotor.homeRequiredIndication OR motorizedSealFlatteners.sealFlattenersHorizontalAxisMotor.Faulted)
														AND readyToRun 
														AND NOT HMIData.faultActive
													THEN
														hmiLight.TurnOn();
													END_IF
													
													
													IF HMIData.stopMachine THEN
														setPassthroughPB := FALSE;
														homeJawPB := FALSE;
														startCycle := FALSE;
														HMIData.initiateCycle := FALSE;
														factoryTestModeKeepCycling := FALSE;
														autoModeKeepCycling := FALSE;
														hmiLight.TurnOff();
													END_IF
													
													IF HMIData.sealBarNotAtTemperature.active THEN
														factoryTestModeKeepCycling := FALSE;
														autoModeKeepCycling := FALSE;
													END_IF
													
													IF bagOpened THEN
														IF NOT bagOpenFingers.CheckIfBagGrabbed(FALSE) THEN
															openedBagWasRemoved.Trigger();
															bagOpened := FALSE;
														END_IF
													END_IF
													
													{region:'Service'}
													IF setPassthroughPB AND NOT homeJawPB THEN
														hmiLight.BlinkSlow();
														motorizedSealFlatteners.sealFlattenersHorizontalAxisMotor.MoveToPositionTorque(2,1000,1000,2000,125);
														state := HEAD_STATES.MovePassthrough;
													END_IF
													IF homeJawPB THEN
														hmiLight.BlinkSlow();
														state := HEAD_STATES.StartHoming;
													END_IF    
													
													IF HMIData.loadPlateService.retractCommand OR HMIData.rearLoadPlateService.retractCommand THEN
														rearLoadPlateRetract.ManualOn();
														HMIData.loadPlateService.retractCommand := FALSE;
														HMIData.rearLoadPlateService.retractCommand := FALSE;
													END_IF                                      
                                                    
													IF HMIData.loadPlateService.extendCommand OR HMIData.rearLoadPlateService.extendCommand THEN
														rearLoadPlateRetract.ManualOff();
														HMIData.loadPlateService.extendCommand := FALSE;
														HMIData.rearLoadPlateService.extendCommand := FALSE;
													END_IF
													
													IF HMIData.loadShelfService.retractCommand THEN
														loadShelfExtend.ManualOn();
														HMIData.loadShelfService.retractCommand := FALSE;
													END_IF                                      
                                                    
													IF HMIData.loadShelfService.extendCommand THEN
														loadShelfExtend.ManualOff();
														HMIData.loadShelfService.extendCommand := FALSE;
													END_IF	

													IF HMIData.forwardLoadPlateService.retractCommand THEN
														forwardLoadPlateRetract.ManualOn();
														HMIData.forwardLoadPlateService.retractCommand := FALSE;
													END_IF                                      
                                                    
													IF HMIData.forwardLoadPlateService.extendCommand THEN
														forwardLoadPlateRetract.ManualOff();
														HMIData.forwardLoadPlateService.extendCommand := FALSE;
													END_IF	 
													
													
														
													IF HMIData.IBDService.retractCommand THEN
														IBD.CloseIBD();
														HMIData.IBDService.retractCommand := FALSE;
													END_IF                                      
                                                    
													IF HMIData.IBDService.extendCommand THEN
														IBD.OpenIBD();
														HMIData.IBDService.extendCommand := FALSE;
													END_IF	
														 
													IF HMIData.funnelService.retractCommand THEN
														funnel.OpenNow();
														HMIData.funnelService.retractCommand := FALSE;
													END_IF                                      
                                                    
													IF HMIData.funnelService.extendCommand THEN
														funnel.CloseNow();
														HMIData.funnelService.extendCommand := FALSE;
													END_IF	
	 													
													IF HMIData.pressureBarService.extendCommand THEN
														pressureBar.OpenJaw();
														HMIData.pressureBarService.extendCommand := FALSE;
													END_IF	
														 
													IF HMIData.pressureBarService.retractCommand THEN
														pressureBar.CloseJaw();
														HMIData.pressureBarService.retractCommand := FALSE;
													END_IF	
														 
													IF HMIData.lpaServicePulse THEN
														LPA.Trigger();
														HMIData.lpaServicePulse := FALSE;
													ELSIF HMIData.lpaServiceOn THEN
														LPA.ManualOn();
														HMIData.lpaServiceOn := FALSE;
													ELSIF HMIData.lpaServiceOff THEN
														LPA.ManualOff();
														HMIData.lpaServiceOff := FALSE;
													END_IF
													
													IF HMIData.vacuumServiceOn THEN
														oVacOn := TRUE;
														HMIData.vacuumServiceOn := FALSE;
													ELSIF HMIData.vacuumServiceOff THEN
														oVacOn := FALSE;
														HMIData.vacuumServiceOff := FALSE;
													END_IF
														 
															  
													IF HMIData.hpaServicePulse THEN
														hpa.Trigger();
														HMIData.hpaServicePulse := FALSE;
													ELSIF hpaServiceOnONS.OSR THEN
														HPA.ManualOn();
													ELSIF hpaServiceOnONS.OSF THEN
														HPA.ManualOff();
													END_IF
													
													IF HMIData.exitConveyorStartDwell THEN
														exitConveyorRun.Trigger();
														HMIData.exitConveyorStartDwell := FALSE;
													ELSIF HMIData.exitConveyorStart OR exitConveyorJogONS.OSR THEN
														exitConveyorRun.ManualOn();
														HMIData.exitConveyorStart := FALSE;
													ELSIF HMIData.exitConveyorStop OR exitConveyorJogONS.OSF THEN
														exitConveyorRun.ManualOff();
														HMIData.exitConveyorStop := FALSE;
													END_IF
													
													IF HMIData.externalExitConveyorStartDwell THEN
														externalExitConveyorRun.Trigger();
														HMIData.externalExitConveyorStartDwell := FALSE;
													ELSIF HMIData.externalExitConveyorStart OR externalExitConveyorJogONS.OSR THEN
														externalExitConveyorRun.ManualOn();
														HMIData.externalExitConveyorStart := FALSE;
													ELSIF HMIData.externalExitConveyorStop OR externalExitConveyorJogONS.OSF THEN
														externalExitConveyorRun.ManualOff();
														HMIData.externalExitConveyorStop := FALSE;
													END_IF
	 
													IF HMIData.sealBarServiceCycle THEN
														sealTimer.PT := TO_TIME(HMIData.sealBarDwell * 1000);
														sealTimer.IN := TRUE;
														IF NOT sealTimer.Q THEN
															oSealBarExtend := TRUE;
															oSealBarRetract := FALSE;
														ELSE 
															sealTimer.IN := FALSE;
															oSealBarExtend := FALSE;
															oSealBarRetract := TRUE;
															HMIData.sealBarCycles.Increment();
															HMIData.sealBarServiceCycle := FALSE;
														END_IF
													ELSIF HMIData.sealBarServiceExtend THEN
														oSealBarExtend := TRUE;
														oSealBarRetract := FALSE;
														HMIData.sealBarServiceExtend := FALSE;
													ELSIF HMIData.sealBarServiceRetract THEN
														oSealBarExtend := FALSE;
														oSealBarRetract := TRUE;
														HMIData.sealBarServiceRetract := FALSE;
													END_IF
														 
													IF HMIData.bagOpenFingersServiceGrab THEN
														bagOpenFingers.Grab();
														HMIData.bagOpenFingersServiceGrab := FALSE;
													ELSIF HMIData.bagOpenFingersServiceRelease THEN
														bagOpenFingers.Release();
														HMIData.bagOpenFingersServiceRelease := FALSE;
													END_IF
		  
													{endregion:'Service'}
                                                    
    HEAD_STATES.SealAndSeparateBag :                // Begin Seal and Separate State machine
													IF enableIBDDeflate THEN
														sealAndSeparateSubState := SEAL_SEPARATE_STATES.BringInIBD;
													ELSE
														sealAndSeparateSubState := SEAL_SEPARATE_STATES.WaitForJawCloseDelay;
													END_IF
													IF printAndApply.enable AND bagOpened THEN
														printAndApply.BeginCycle();
													END_IF
													filler.BaggerCycleInitiated();
                                                    HMIData.inCycle := TRUE;
													HMIData.airFilterClean.Increment();
													HMIData.baggerCycles.Increment();
													IF funnel.enable THEN
														funnel.CloseNow();
													END_IF
													
                                                    state := HEAD_STATES.SealingAndSeparatingBag;
                                                    
                
    HEAD_STATES.SealingAndSeparatingBag :            IF sealAndSeparateSubState = SEAL_SEPARATE_STATES.Done THEN
                                                        state := HEAD_STATES.SealedAndSeparatedBag;
                                                        sealAndSeparateSubState := SEAL_SEPARATE_STATES.Idle;
                                                    END_IF    

    HEAD_STATES.SealedAndSeparatedBag :                state := HEAD_STATES.ReleaseAndFeedBag;                                    
                                                    
    HEAD_STATES.ReleaseAndFeedBag :                    // Open the jaw and release the bag
                                                    releaseAndFeedSubState := RELEASE_FEED_STATES.MoveJawOutAndDropBag;
                                                    state := HEAD_STATES.ReleasingAndFeedingBag;
                                                    
    HEAD_STATES.ReleasingAndFeedingBag :            // 
                                                    IF releaseAndFeedSubState = RELEASE_FEED_STATES.Done THEN
                                                        state := HEAD_STATES.ReleasedAndFedBag;
                                                        releaseAndFeedSubState := RELEASE_FEED_STATES.Idle;
                                                    END_IF
                                                    
    HEAD_STATES.ReleasedAndFedBag :                    // 
                                                    {warning 'TODO: change this counting logic to account for MSF'}
                                                    IF enableBatch THEN
                                                        batchCount := batchCount + 1;
                                                    END_IF
  
                                                    IF Globals.enableDryCycle THEN
                                                        Globals.dryCycleCount := Globals.dryCycleCount + 1;     
                                                    ELSE
                                                        Globals.bagsMadeCount := Globals.bagsMadeCount + 1; 
                                                    END_IF
													IF enableBagOpen THEN
                                                        state := HEAD_STATES.OpenBag;
                                                    ELSE
                                                        state := HEAD_STATES.FinishCycle;
                                                    END_IF
                                                    
                                                            
                                                    
                                
    HEAD_STATES.OpenBag :                            // Close jaw to grab the bag
                                                    openBagSubState := BAG_OPEN_ASSIST_STATES.MoveJawIn;
                                                    state := HEAD_STATES.OpeningBag;
                                                    
                                                    
    HEAD_STATES.OpeningBag :                        // Open jaw and grab onto the bag
                                                    IF openBagSubState = BAG_OPEN_ASSIST_STATES.Done THEN
                                                        state := HEAD_STATES.OpenedBag;
                                                        openBagSubState := BAG_OPEN_ASSIST_STATES.Idle;
													ELSIF openBagSubState = BAG_OPEN_ASSIST_STATES.FeedNewBag THEN
														state := HEAD_STATES.SealAndSeparateBag;
														openBagSubState := BAG_OPEN_ASSIST_STATES.Idle;
                                                    END_IF
                                                    
    HEAD_STATES.OpenedBag :                            // Move fingers in and to bag holding and reset cycle
                                                    IF (motorizedSealFlatteners.state = SEAL_FLATTENER_STATES.Idle OR NOT motorizedSealFlatteners.enable) //OR bagFailedToOpen
														 AND pressureBar.state = PRESSURE_BAR_STATES.Idle THEN
														state := HEAD_STATES.FinishCycle;
                                                    END_IF
	HEAD_STATES.FinishCycle :			//
													finishCycleSubState := FINISH_CYCLE_STATES.Start;
													state := HEAD_STATES.FinishingCycle;
	HEAD_STATES.FinishingCycle : 		//
													IF finishCycleSubState = FINISH_CYCLE_STATES.Done THEN
														state := HEAD_STATES.FinishedCycle;
														finishCycleSubState := FINISH_CYCLE_STATES.Idle;
													END_IF
	HEAD_STATES.FinishedCycle :			//
											HMIData.bagsMade.Increment();
											HMIData.resettableBagsMade.Increment();
                                            state := HEAD_STATES.Idle;
											filler.BaggerCycledAndReady();
											cycleTime := (TIME_TO_REAL(cycleTimer.ET) / 1000); 
											cycleTimer.IN := FALSE;
											IF HMIData.averageCycleTime = 0 THEN
												HMIData.averageCycleTime := cycleTime;
											ELSE
												HMIData.averageCycleTime := (cycleTime + HMIData.averageCycleTime) / 2;
											END_IF
											HMIData.inCycle := FALSE;
											//bagFailedToOpen := FALSE;
											
											IF HMIData.autoEnable AND NOT HMIData.stopMachine THEN
												autoModeKeepCycling := TRUE;
											END_IF
											
											IF HMIData.factoryTestMode AND NOT HMIData.stopMachine THEN
												IF (HMIData.bagsMade.count >= 1000) THEN
													factoryTestModeKeepCycling := FALSE;
													HMIData.factoryTestMode := FALSE;
												ELSE
													factoryTestModeKeepCycling := TRUE;
												END_IF
											END_IF	
	HEAD_STATES.StartReset 	:			// Reset all 
	
	HEAD_STATES.Resetting : 

										
    HEAD_STATES.StartHoming :            // 
											IF allMotorCommsGood THEN
												motorizedSealFlatteners.sealFlattenersHorizontalAxisMotor.faults.notHomed.Ack();
												IF pressureBar.homeRequired THEN
													pressureBar.HomeNow();
												ELSE
													pressureBar.OpenJaw();
												END_IF
												IF IBD.homeRequired THEN
													IF NOT enableLabelSideUp THEN
														rearLoadPlateRetract.ManualOn();
													END_IF
													IBD.HomeNow();
												ELSE
													IBD.OpenIBD();
												END_IF
												
                                            	state := HEAD_STATES.Homing; 
											END_IF
                                                                                   
    
    HEAD_STATES.Homing :                // 
                                            //IF NOT pressureBar.homeRequired AND (NOT IBD.homeRequired OR NOT IBD.enable) THEN
											IF pressureBar.pressureBarOpen AND (NOT IBD.Ready OR NOT IBD.enable) THEN
                                                state := HEAD_STATES.HomingComplete;
												rearLoadPlateRetract.ManualOff();   
												IF motorizedSealFlatteners.sealFlattenersHorizontalAxisMotor.HomeRequired AND HMIData.sealFlattenersSelection = SealFlattenerSelection.MotorizedSealFlatteners THEN
													motorizedSealFlatteners.sealFlattenersHorizontalAxisMotor.HomeNow();
													motorizedSealFlatteners.sealFlattenersVerticalAxis.Retract();
												END_IF    
                                            END_IF
                                            
    HEAD_STATES.HomingComplete :        // 
											IF NOT motorizedSealFlatteners.sealFlattenersHorizontalAxisMotor.HomeRequired THEN
												 homeJawPB := FALSE;
												state := HEAD_STATES.Idle;
												//HMIData.passthroughSetting := 6.0;
												setPassthroughPB := TRUE;
											END_IF
                                           
    
    HEAD_STATES.MovePassthrough :        // 
                                            pressureBar.OpenJaw();
											IBD.OpenIBD();
											
                                            state := HEAD_STATES.MovingPassthrough;
    
    HEAD_STATES.MovingPassthrough :    		IF pressureBar.pressureBarOpen AND IBD.IBDOpen THEN
                                                state := HEAD_STATES.MovedPassthrough;     
												motorizedSealFlatteners.sealFlattenersHorizontalAxisMotor.MoveToPositionTorque(HMIData.bagWidth,1000,1000,1000,25);
                                            END_IF
                                            
    HEAD_STATES.MovedPassthrough :        // 
                                            //pressureBar.AutoDoneMovingPassthrough();
                                            state := HEAD_STATES.Idle;
											setPassthroughPB := FALSE;
                                                    
    HEAD_STATES.Fault :                     hmiLight.TurnOff();
											HMIData.inCycle := FALSE;
											cycleTimer.IN := FALSE;
											bagDelivery.bagFeedMasterMotor.SetRearMotorToEncoderFollowing();
											sealAndSeparateSubState := SEAL_SEPARATE_STATES.Idle;
											releaseAndFeedSubState := RELEASE_FEED_STATES.Idle;
											openBagSubState := BAG_OPEN_ASSIST_STATES.Idle;
											finishCycleSubState := FINISH_CYCLE_STATES.Idle;
											oVacOn := FALSE;
											filler.Reset();
											LPA.ManualOff();
											//IBD.Reset();
											exitConveyorRun.Reset();
											externalExitConveyorRun.Reset();
											oRunPrinterRibbonUnwindMotor := FALSE;
											setPassthroughPB := FALSE;
											homeJawPB := FALSE;
											startCycle := FALSE;
											HMIData.initiateCycle := FALSE;
											factoryTestModeKeepCycling := FALSE;
											autoModeKeepCycling := FALSE;
											pressureBarCloseDelay.IN := FALSE;
											//bagOpened := FALSE;
                                                    
END_CASE

CASE sealAndSeparateSubState OF
    SEAL_SEPARATE_STATES.Idle : 
	
	SEAL_SEPARATE_STATES.BringInIBD : 				// Bring in IBD if enabled
													IF enableIBDDeflate THEN
														IBD.CloseIBD();
													END_IF 
													
													sealAndSeparateSubState := SEAL_SEPARATE_STATES.WaitForJawCloseDelay;
	
	SEAL_SEPARATE_STATES.WaitForJawCloseDelay : 	// Wait for jaw close delay. 
													IF pressureBar.enable THEN
														LPA.ManualOff();
														pressureBarCloseDelay.IN := TRUE;
														IF (pressureBarCloseDelay.Q OR HMIData.pressureBarCloseDelay = 0) 
															AND (funnel.closed OR NOT funnel.enable)
															THEN
															sealAndSeparateSubState := SEAL_SEPARATE_STATES.MoveJawIn;
															pressureBarCloseDelay.IN := FALSE;
														END_IF
                                                    ELSE 
                                                        sealAndSeparateSubState := SEAL_SEPARATE_STATES.ReverseBag;
                                                    END_IF
        
    SEAL_SEPARATE_STATES.MoveJawIn :                // Perform actions as enabled - close jaw and move flatteners out. If jaw is disabled then go right to reverse bag
                                                    IF motorizedSealFlatteners.enable THEN
                                                        motorizedSealFlatteners.AutoMoveOut();
                                                    END_IF
                                                    
													pressureBar.CloseJaw();
                                                    sealAndSeparateSubState := SEAL_SEPARATE_STATES.MovingJawIn;
                                                    
                                                    
                                                    
                                                    
                                                    
    SEAL_SEPARATE_STATES.MovingJawIn :                // If Jaw is in and flatteners out then move on
                                                    IF (motorizedSealFlatteners.state = SEAL_FLATTENER_STATES.MovedFlattenersOut OR NOT motorizedSealFlatteners.enable) 
                                                        AND (pressureBar.clamped OR NOT pressureBar.enable)
                                                        THEN
                                                            sealAndSeparateSubState := SEAL_SEPARATE_STATES.MovedJawIn;    
                                                    END_IF
                                                                
    SEAL_SEPARATE_STATES.MovedJawIn :                // Will add sealing logic here
                                                    sealAndSeparateSubState := SEAL_SEPARATE_STATES.ReverseBag;
                                                    
    SEAL_SEPARATE_STATES.ReverseBag :                // Reverse bag if bag delivery enabled, otherwise open jaw
													//IBD.OpenFull();
                                                    IF bagDelivery.enable THEN
                                                        bagDelivery.AutoReverseBag();
                                                        sealAndSeparateSubState := SEAL_SEPARATE_STATES.ReversingBag;
                                                    ELSE sealAndSeparateSubState := SEAL_SEPARATE_STATES.Done;    
                                                    END_IF
                                                                    
    SEAL_SEPARATE_STATES.ReversingBag :                // 
													IF NOT HMIData.separateBeforeSeal THEN
														sealTimer.PT := TO_TIME(HMIData.sealBarDwell * 1000);
														sealTimer.IN := TRUE;
														IF NOT sealTimer.Q THEN
															oSealBarExtend := TRUE;
															oSealBarRetract := FALSE;
														ELSE 
															
															oSealBarExtend := FALSE;
															oSealBarRetract := TRUE;
															
														END_IF
													END_IF

                                                    IF (motorizedSealFlatteners.state = SEAL_FLATTENER_STATES.MovedFlattenersOut OR NOT motorizedSealFlatteners.enable) 
                                                        AND (pressureBar.clamped OR NOT pressureBar.enable)
                                                        AND (bagDelivery.state = BAG_DELIVERY_STATES.ReverseDone OR NOT bagDelivery.enable)
														AND (sealTimer.Q OR HMIData.separateBeforeSeal)
                                                        THEN
															IF NOT HMIData.separateBeforeSeal THEN
																HMIData.sealBarCycles.Increment();
															END_IF
															
															sealTimer.IN := FALSE;
                                                            sealAndSeparateSubState := SEAL_SEPARATE_STATES.Reversedbag;
                                                    END_IF
    SEAL_SEPARATE_STATES.Reversedbag :                // 
                                                    sealAndSeparateSubState := SEAL_SEPARATE_STATES.SealBag;
													
	SEAL_SEPARATE_STATES.SealBag:					
													IF HMIData.separateBeforeSeal THEN
														sealTimer.PT := TO_TIME(HMIData.sealBarDwell * 1000);
														sealTimer.IN := TRUE;
														IF NOT sealTimer.Q THEN
															oSealBarExtend := TRUE;
															oSealBarRetract := FALSE;
														ELSE 
															sealTimer.IN := FALSE;
															oSealBarExtend := FALSE;
															oSealBarRetract := TRUE;
															HMIData.sealBarCycles.Increment();
															sealAndSeparateSubState := SEAL_SEPARATE_STATES.Done;
														END_IF
													ELSE
														sealAndSeparateSubState := SEAL_SEPARATE_STATES.Done;
													END_IF
													
																				
                                                    
    SEAL_SEPARATE_STATES.Done :                        // 
                                                    
